LIN {X 0,Y 162.49,Z 738.182,A -85,B 0,C 180,E1 -25157.336,E2 -25157.336} C_VEL
LIN {X 0,Y 169.841,Z 726.293,A -85,B 0,C 180,E1 -25160.422,E2 -25160.422} C_VEL
LIN {X 0,Y 176.479,Z 714.157,A -85,B 0,C 180,E1 -25162.799,E2 -25162.799} C_VEL
LIN {X 0,Y 182.421,Z 701.363,A -85,B 0,C 180,E1 -25164.776,E2 -25164.776} C_VEL
LIN {X 0,Y 187.765,Z 687.719,A -85,B 0,C 180,E1 -25166.394,E2 -25166.394} C_VEL
LIN {X 0,Y 192.387,Z 673.366,A -85,B 0,C 180,E1 -25167.653,E2 -25167.653} C_VEL
LIN {X 0,Y 195.327,Z 661.656,A -85,B 0,C 180,E1 -25168.438,E2 -25168.438} C_VEL
LIN {X 0,Y 188.681,Z 668.85,A -85,B 0,C 180,E1 -25170.426,E2 -25170.426} C_VEL
LIN {X 0,Y 182.829,Z 674.036,A -85,B 0,C 180,E1 -25172.53,E2 -25172.53} C_VEL
LIN {X 0,Y 181.051,Z 675.427,A -85,B 0,C 180,E1 -25173.234,E2 -25173.234} C_VEL
LIN {X 0,Y 174.563,Z 681.994,A -85,B 0,C 180,E1 -25175.551,E2 -25175.551} C_VEL
LIN {X 0,Y 168.965,Z 686.875,A -85,B 0,C 180,E1 -25178.016,E2 -25178.016} C_VEL
LIN {X 0,Y 165.167,Z 689.589,A -85,B 0,C 180,E1 -25180.098,E2 -25180.098} C_VEL
LIN {X 0,Y 163.165,Z 690.902,A -85,B 0,C 180,E1 -25181.38,E2 -25181.38} C_VEL
LIN {X 0,Y 156.436,Z 696.804,A -85,B 0,C 180,E1 -25185.483,E2 -25185.483} C_VEL
LIN {X 0,Y 152.151,Z 700.127,A -85,B 0,C 180,E1 -25189.352,E2 -25189.352} C_VEL
LIN {X 0,Y 149.893,Z 701.971,A -85,B 0,C 180,E1 -25191.914,E2 -25191.914} C_VEL
LIN {X 0,Y 147.571,Z 704.34,A -85,B 0,C 180,E1 -25194.534,E2 -25194.534} C_VEL
LIN {X 0,Y 145.899,Z 706.177,A -85,B 0,C 180,E1 -25197.239,E2 -25197.239} C_VEL
LIN {X 0,Y 143.539,Z 710.381,A -85,B 0,C 180,E1 -25205.619,E2 -25205.619} C_VEL
LIN {X 0,Y 143.347,Z 711.889,A -85,B 0,C 180,E1 -25208.458,E2 -25208.458} C_VEL
LIN {X 0,Y 144.725,Z 713.835,A -85,B 0,C 180,E1 -25214.052,E2 -25214.052} C_VEL
LIN {X 0,Y 149.356,Z 716.433,A -85,B 0,C 180,E1 -25222.113,E2 -25222.113} C_VEL
LIN {X 0,Y 154.656,Z 717.177,A -85,B 0,C 180,E1 -25227.028,E2 -25227.028} C_VEL
LIN {X 0,Y 161.315,Z 717.454,A -85,B 0,C 180,E1 -25231.52,E2 -25231.52} C_VEL
LIN {X 0,Y 168.975,Z 717.586,A -85,B 0,C 180,E1 -25235.611,E2 -25235.611} C_VEL
LIN {X 0,Y 173.986,Z 717.219,A -85,B 0,C 180,E1 -25237.718,E2 -25237.718} C_VEL
LIN {X 0,Y 173.679,Z 718.782,A -85,B 0,C 180,E1 -25238.224,E2 -25238.224} C_VEL
LIN {X 0,Y 167.056,Z 730.388,A -85,B 0,C 180,E1 -25240.773,E2 -25240.773} C_VEL
LIN {X 0,Y 160.359,Z 740.731,A -85,B 0,C 180,E1 -25243.681,E2 -25243.681} C_VEL
LIN {X 0,Y 153.45,Z 750.501,A -85,B 0,C 180,E1 -25247.278,E2 -25247.278} C_VEL
LIN {X 0,Y 147.243,Z 758.709,A -85,B 0,C 180,E1 -25251.245,E2 -25251.245} C_VEL
LIN {X 0,Y 144.176,Z 761.795,A -85,B 0,C 180,E1 -25252.828,E2 -25252.828} C_VEL
LIN {X 0,Y 137.87,Z 766.464,A -85,B 0,C 180,E1 -25255.293,E2 -25255.293} C_VEL
LIN {X 0,Y 131.777,Z 770.674,A -85,B 0,C 180,E1 -25258.095,E2 -25258.095} C_VEL
LIN {X 0,Y 129.133,Z 772.932,A -85,B 0,C 180,E1 -25260.184,E2 -25260.184} C_VEL
LIN {X 0,Y 124.453,Z 778.128,A -85,B 0,C 180,E1 -25266.71,E2 -25266.71} C_VEL
LIN {X 0,Y 121.396,Z 781.651,A -85,B 0,C 180,E1 -25273.169,E2 -25273.169} C_VEL
LIN {X 0,Y 119.749,Z 783.963,A -85,B 0,C 180,E1 -25279.854,E2 -25279.854} C_VEL
LIN {X 0,Y 119.228,Z 785.118,A -85,B 0,C 180,E1 -25286.615,E2 -25286.615} C_VEL
LIN {X 0,Y 119.279,Z 785.267,A -85,B 0,C 180,E1 -25289.995,E2 -25289.995} C_VEL
LIN {X 0,Y 119.386,Z 784.666,A -85,B 0,C 180,E1 -25296.756,E2 -25296.756} C_VEL
LIN {X 0,Y 120.432,Z 782.915,A -85,B 0,C 180,E1 -25303.493,E2 -25303.493} C_VEL
LIN {X 0,Y 122.725,Z 779.989,A -85,B 0,C 180,E1 -25310.09,E2 -25310.09} C_VEL
LIN {X 0,Y 126.443,Z 775.815,A -85,B 0,C 180,E1 -25316.396,E2 -25316.396} C_VEL
LIN {X 0,Y 131.402,Z 770.282,A -85,B 0,C 180,E1 -25322.327,E2 -25322.327} C_VEL
LIN {X 0,Y 137.622,Z 763.238,A -85,B 0,C 180,E1 -25327.787,E2 -25327.787} C_VEL
LIN {X 0,Y 144.102,Z 755.689,A -85,B 0,C 180,E1 -25332.107,E2 -25332.107} C_VEL
LIN {X 0,Y 149.999,Z 747.998,A -85,B 0,C 180,E1 -25335.597,E2 -25335.597} C_VEL
LIN {X 0,Y 157.779,Z 737.318,A -85,B 0,C 180,E1 -25339.214,E2 -25339.214} C_VEL
LIN {X 0,Y 165.444,Z 725.295,A -85,B 0,C 180,E1 -25342.289,E2 -25342.289} C_VEL
LIN {X 0,Y 172.284,Z 713.017,A -85,B 0,C 180,E1 -25344.665,E2 -25344.665} C_VEL
LIN {X 0,Y 178.544,Z 699.747,A -85,B 0,C 180,E1 -25346.657,E2 -25346.657} C_VEL
LIN {X 0,Y 183.943,Z 686.095,A -85,B 0,C 180,E1 -25348.217,E2 -25348.217} C_VEL
LIN {X 0,Y 188.689,Z 671.315,A -85,B 0,C 180,E1 -25349.458,E2 -25349.458} C_VEL
LIN {X 0,Y 192.33,Z 656.608,A -85,B 0,C 180,E1 -25350.334,E2 -25350.334} C_VEL
LIN {X 0,Y 194.901,Z 641.487,A -85,B 0,C 180,E1 -25350.971,E2 -25350.971} C_VEL
LIN {X 0,Y 201.625,Z 569.905,A -85,B 0,C 180,E1 -25352.853,E2 -25352.853} C_VEL
LIN {X 0,Y 204.85,Z 533.822,A -85,B 0,C 180,E1 -25353.826,E2 -25353.826} C_VEL
LIN {X 0,Y 204.843,Z 524.765,A -85,B 0,C 180,E1 -25354.546,E2 -25354.546} C_VEL
LIN {X 0,Y 201.445,Z 518.518,A -85,B 0,C 180,E1 -25357.23,E2 -25357.23} C_VEL
LIN {X 0,Y 196.969,Z 511.105,A -85,B 0,C 180,E1 -25361.404,E2 -25361.404} C_VEL
LIN {X 0,Y 194.313,Z 507.036,A -85,B 0,C 180,E1 -25364.456,E2 -25364.456} C_VEL
LIN {X 0,Y 190.943,Z 502.129,A -85,B 0,C 180,E1 -25369.663,E2 -25369.663} C_VEL
LIN {X 0,Y 189.493,Z 500.135,A -85,B 0,C 180,E1 -25373.077,E2 -25373.077} C_VEL
LIN {X 0,Y 188.395,Z 499.148,A -85,B 0,C 180,E1 -25377.862,E2 -25377.862} C_VEL
LIN {X 0,Y 188.294,Z 499.346,A -85,B 0,C 180,E1 -25381.07,E2 -25381.07} C_VEL
LIN {X 0,Y 188.705,Z 500.765,A -85,B 0,C 180,E1 -25384.564,E2 -25384.564} C_VEL
LIN {X 0,Y 190.134,Z 504.27,A -85,B 0,C 180,E1 -25389.173,E2 -25389.173} C_VEL
LIN {X 0,Y 192.543,Z 509.234,A -85,B 0,C 180,E1 -25393.631,E2 -25393.631} C_VEL
LIN {X 0,Y 195.143,Z 514.935,A -85,B 0,C 180,E1 -25397.172,E2 -25397.172} C_VEL
LIN {X 0,Y 197.823,Z 520.849,A -85,B 0,C 180,E1 -25400.131,E2 -25400.131} C_VEL
LIN {X 0,Y 200.646,Z 527.803,A -85,B 0,C 180,E1 -25402.849,E2 -25402.849} C_VEL
LIN {X 0,Y 203.756,Z 536.057,A -85,B 0,C 180,E1 -25405.5,E2 -25405.5} C_VEL
LIN {X 0,Y 204.496,Z 538.387,A -85,B 0,C 180,E1 -25406.111,E2 -25406.111} C_VEL
LIN {X 0,Y 204.503,Z 541.924,A -85,B 0,C 180,E1 -25406.39,E2 -25406.39} C_VEL
LIN {X 0,Y 195.309,Z 640.75,A -85,B 0,C 180,E1 -25408.979,E2 -25408.979} C_VEL
LIN {X 0,Y 192.93,Z 655.292,A -85,B 0,C 180,E1 -25409.583,E2 -25409.583} C_VEL
LIN {X 0,Y 189.481,Z 669.768,A -85,B 0,C 180,E1 -25410.425,E2 -25410.425} C_VEL
LIN {X 0,Y 185.336,Z 682.994,A -85,B 0,C 180,E1 -25411.446,E2 -25411.446} C_VEL
LIN {X 0,Y 180.038,Z 696.994,A -85,B 0,C 180,E1 -25412.945,E2 -25412.945} C_VEL
LIN {X 0,Y 174.103,Z 710.142,A -85,B 0,C 180,E1 -25414.817,E2 -25414.817} C_VEL
LIN {X 0,Y 167.333,Z 722.659,A -85,B 0,C 180,E1 -25417.067,E2 -25417.067} C_VEL
LIN {X 0,Y 161.275,Z 732.55,A -85,B 0,C 180,E1 -25419.337,E2 -25419.337} C_VEL
LIN {X 0,Y 154.403,Z 742.63,A -85,B 0,C 180,E1 -25422.305,E2 -25422.305} C_VEL
LIN {X 0,Y 146.952,Z 752.624,A -85,B 0,C 180,E1 -25426.215,E2 -25426.215} C_VEL
LIN {X 0,Y 140.359,Z 760.636,A -85,B 0,C 180,E1 -25430.333,E2 -25430.333} C_VEL
LIN {X 0,Y 134.43,Z 767.397,A -85,B 0,C 180,E1 -25434.901,E2 -25434.901} C_VEL
LIN {X 0,Y 128.273,Z 774.274,A -85,B 0,C 180,E1 -25441.239,E2 -25441.239} C_VEL
LIN {X 0,Y 124.469,Z 778.502,A -85,B 0,C 180,E1 -25446.724,E2 -25446.724} C_VEL
LIN {X 0,Y 121.342,Z 782.047,A -85,B 0,C 180,E1 -25453.172,E2 -25453.172} C_VEL
LIN {X 0,Y 119.681,Z 784.387,A -85,B 0,C 180,E1 -25459.859,E2 -25459.859} C_VEL
LIN {X 0,Y 119.151,Z 785.575,A -85,B 0,C 180,E1 -25466.624,E2 -25466.624} C_VEL
LIN {X 0,Y 119.227,Z 785.732,A -85,B 0,C 180,E1 -25470.005,E2 -25470.005} C_VEL
LIN {X 0,Y 119.292,Z 785.153,A -85,B 0,C 180,E1 -25476.772,E2 -25476.772} C_VEL
LIN {X 0,Y 120.374,Z 783.432,A -85,B 0,C 180,E1 -25483.511,E2 -25483.511} C_VEL
LIN {X 0,Y 122.702,Z 780.532,A -85,B 0,C 180,E1 -25490.105,E2 -25490.105} C_VEL
LIN {X 0,Y 126.437,Z 776.387,A -85,B 0,C 180,E1 -25496.408,E2 -25496.408} C_VEL
LIN {X 0,Y 131.398,Z 770.896,A -85,B 0,C 180,E1 -25502.34,E2 -25502.34} C_VEL
LIN {X 0,Y 137.603,Z 763.906,A -85,B 0,C 180,E1 -25507.804,E2 -25507.804} C_VEL
LIN {X 0,Y 144.095,Z 756.412,A -85,B 0,C 180,E1 -25512.121,E2 -25512.121} C_VEL
LIN {X 0,Y 151.1,Z 747.379,A -85,B 0,C 180,E1 -25516.137,E2 -25516.137} C_VEL
LIN {X 0,Y 157.743,Z 738.16,A -85,B 0,C 180,E1 -25519.241,E2 -25519.241} C_VEL
LIN {X 0,Y 165.391,Z 726.268,A -85,B 0,C 180,E1 -25522.325,E2 -25522.325} C_VEL
LIN {X 0,Y 172.271,Z 714.129,A -85,B 0,C 180,E1 -25524.684,E2 -25524.684} C_VEL
LIN {X 0,Y 178.649,Z 700.77,A -85,B 0,C 180,E1 -25526.722,E2 -25526.722} C_VEL
LIN {X 0,Y 184.265,Z 686.688,A -85,B 0,C 180,E1 -25528.345,E2 -25528.345} C_VEL
LIN {X 0,Y 187.983,Z 675.523,A -85,B 0,C 180,E1 -25529.309,E2 -25529.309} C_VEL
LIN {X 0,Y 187.675,Z 675.519,A -85,B 0,C 180,E1 -25529.468,E2 -25529.468} C_VEL
LIN {X 0,Y 180.025,Z 681.759,A -85,B 0,C 180,E1 -25532.065,E2 -25532.065} C_VEL
LIN {X 0,Y 173.593,Z 687.748,A -85,B 0,C 180,E1 -25534.2,E2 -25534.2} C_VEL
LIN {X 0,Y 167.992,Z 692.21,A -85,B 0,C 180,E1 -25536.451,E2 -25536.451} C_VEL
LIN {X 0,Y 163.738,Z 695.116,A -85,B 0,C 180,E1 -25538.602,E2 -25538.602} C_VEL
LIN {X 0,Y 159.607,Z 697.882,A -85,B 0,C 180,E1 -25540.95,E2 -25540.95} C_VEL
LIN {X 0,Y 154.095,Z 702.368,A -85,B 0,C 180,E1 -25544.118,E2 -25544.118} C_VEL
LIN {X 0,Y 148.318,Z 706.43,A -85,B 0,C 180,E1 -25549.074,E2 -25549.074} C_VEL
LIN {X 0,Y 143.513,Z 710.534,A -85,B 0,C 180,E1 -25554.379,E2 -25554.379} C_VEL
LIN {X 0,Y 140.677,Z 713.581,A -85,B 0,C 180,E1 -25560,E2 -25560} C_VEL
LIN {X 0,Y 139.122,Z 717.695,A -85,B 0,C 180,E1 -25568.716,E2 -25568.716} C_VEL
LIN {X 0,Y 140.542,Z 719.536,A -85,B 0,C 180,E1 -25574.479,E2 -25574.479} C_VEL
LIN {X 0,Y 145.295,Z 722.025,A -85,B 0,C 180,E1 -25582.765,E2 -25582.765} C_VEL
LIN {X 0,Y 150.733,Z 722.733,A -85,B 0,C 180,E1 -25587.791,E2 -25587.791} C_VEL
LIN {X 0,Y 161.277,Z 723.193,A -85,B 0,C 180,E1 -25594.507,E2 -25594.507} C_VEL
LIN {X 0,Y 166.326,Z 723.054,A -85,B 0,C 180,E1 -25596.909,E2 -25596.909} C_VEL
LIN {X 0,Y 166.11,Z 724.465,A -85,B 0,C 180,E1 -25597.481,E2 -25597.481} C_VEL
LIN {X 0,Y 158.98,Z 735.806,A -85,B 0,C 180,E1 -25600.304,E2 -25600.304} C_VEL
LIN {X 0,Y 152.197,Z 745.306,A -85,B 0,C 180,E1 -25603.335,E2 -25603.335} C_VEL
LIN {X 0,Y 145.117,Z 754.626,A -85,B 0,C 180,E1 -25607.306,E2 -25607.306} C_VEL
LIN {X 0,Y 138.553,Z 762.37,A -85,B 0,C 180,E1 -25611.578,E2 -25611.578} C_VEL
LIN {X 0,Y 132.923,Z 768.782,A -85,B 0,C 180,E1 -25616.273,E2 -25616.273} C_VEL
LIN {X 0,Y 129.133,Z 772.932,A -85,B 0,C 180,E1 -25620.184,E2 -25620.184} C_VEL
LIN {X 0,Y 126.612,Z 775.054,A -85,B 0,C 180,E1 -25622.385,E2 -25622.385} C_VEL
LIN {X 0,Y 121.161,Z 778.137,A -85,B 0,C 180,E1 -25625.944,E2 -25625.944} C_VEL
LIN {X 0,Y 116.992,Z 780.194,A -85,B 0,C 180,E1 -25629.05,E2 -25629.05} C_VEL
LIN {X 0,Y 114.808,Z 781.484,A -85,B 0,C 180,E1 -25631.694,E2 -25631.694} C_VEL
LIN {X 0,Y 114.384,Z 781.855,A -85,B 0,C 180,E1 -25632.64,E2 -25632.64} C_VEL
LIN {X 0,Y 112.741,Z 783.977,A -85,B 0,C 180,E1 -25639.216,E2 -25639.216} C_VEL
LIN {X 0,Y 112.135,Z 785.132,A -85,B 0,C 180,E1 -25646.401,E2 -25646.401} C_VEL
LIN {X 0,Y 112.198,Z 785.281,A -85,B 0,C 180,E1 -25649.994,E2 -25649.994} C_VEL
LIN {X 0,Y 112.307,Z 784.679,A -85,B 0,C 180,E1 -25657.184,E2 -25657.184} C_VEL
LIN {X 0,Y 113.5,Z 782.929,A -85,B 0,C 180,E1 -25664.335,E2 -25664.335} C_VEL
LIN {X 0,Y 116.051,Z 780.003,A -85,B 0,C 180,E1 -25671.301,E2 -25671.301} C_VEL
LIN {X 0,Y 120.062,Z 775.829,A -85,B 0,C 180,E1 -25677.917,E2 -25677.917} C_VEL
LIN {X 0,Y 125.406,Z 770.296,A -85,B 0,C 180,E1 -25684.078,E2 -25684.078} C_VEL
LIN {X 0,Y 132.036,Z 763.253,A -85,B 0,C 180,E1 -25689.691,E2 -25689.691} C_VEL
LIN {X 0,Y 138.874,Z 755.704,A -85,B 0,C 180,E1 -25694.088,E2 -25694.088} C_VEL
LIN {X 0,Y 143.97,Z 749.356,A -85,B 0,C 180,E1 -25697.067,E2 -25697.067} C_VEL
LIN {X 0,Y 152.012,Z 738.949,A -85,B 0,C 180,E1 -25700.744,E2 -25700.744} C_VEL
LIN {X 0,Y 159.294,Z 728.252,A -85,B 0,C 180,E1 -25703.621,E2 -25703.621} C_VEL
LIN {X 0,Y 166.324,Z 716.568,A -85,B 0,C 180,E1 -25706.014,E2 -25706.014} C_VEL
LIN {X 0,Y 172.742,Z 704.08,A -85,B 0,C 180,E1 -25708.013,E2 -25708.013} C_VEL
LIN {X 0,Y 178.241,Z 691.413,A -85,B 0,C 180,E1 -25709.593,E2 -25709.593} C_VEL
LIN {X 0,Y 183.097,Z 678.132,A -85,B 0,C 180,E1 -25710.829,E2 -25710.829} C_VEL
LIN {X 0,Y 187.313,Z 663.497,A -85,B 0,C 180,E1 -25711.842,E2 -25711.842} C_VEL
LIN {X 0,Y 190.521,Z 648.344,A -85,B 0,C 180,E1 -25712.568,E2 -25712.568} C_VEL
LIN {X 0,Y 192.614,Z 632.59,A -85,B 0,C 180,E1 -25713.075,E2 -25713.075} C_VEL
LIN {X 0,Y 200.135,Z 552.217,A -85,B 0,C 180,E1 -25715.147,E2 -25715.147} C_VEL
LIN {X 0,Y 201.753,Z 534.762,A -85,B 0,C 180,E1 -25715.606,E2 -25715.606} C_VEL
LIN {X 0,Y 201.757,Z 529.052,A -85,B 0,C 180,E1 -25716.092,E2 -25716.092} C_VEL
LIN {X 0,Y 198.348,Z 522.844,A -85,B 0,C 180,E1 -25719.044,E2 -25719.044} C_VEL
LIN {X 0,Y 194.916,Z 516.851,A -85,B 0,C 180,E1 -25722.593,E2 -25722.593} C_VEL
LIN {X 0,Y 192.637,Z 513.263,A -85,B 0,C 180,E1 -25725.439,E2 -25725.439} C_VEL
LIN {X 0,Y 189.566,Z 508.606,A -85,B 0,C 180,E1 -25730.666,E2 -25730.666} C_VEL
LIN {X 0,Y 188.45,Z 507.051,A -85,B 0,C 180,E1 -25733.576,E2 -25733.576} C_VEL
LIN {X 0,Y 187.532,Z 506.19,A -85,B 0,C 180,E1 -25737.852,E2 -25737.852} C_VEL
LIN {X 0,Y 187.425,Z 506.417,A -85,B 0,C 180,E1 -25741.075,E2 -25741.075} C_VEL
LIN {X 0,Y 187.824,Z 507.961,A -85,B 0,C 180,E1 -25744.586,E2 -25744.586} C_VEL
LIN {X 0,Y 189.081,Z 511.235,A -85,B 0,C 180,E1 -25748.82,E2 -25748.82} C_VEL
LIN {X 0,Y 191.124,Z 515.753,A -85,B 0,C 180,E1 -25752.881,E2 -25752.881} C_VEL
LIN {X 0,Y 193.413,Z 521.078,A -85,B 0,C 180,E1 -25756.255,E2 -25756.255} C_VEL
LIN {X 0,Y 195.988,Z 527.127,A -85,B 0,C 180,E1 -25759.312,E2 -25759.312} C_VEL
LIN {X 0,Y 198.545,Z 533.898,A -85,B 0,C 180,E1 -25761.956,E2 -25761.956} C_VEL
LIN {X 0,Y 201.363,Z 541.93,A -85,B 0,C 180,E1 -25764.538,E2 -25764.538} C_VEL
LIN {X 0,Y 196.477,Z 594.889,A -85,B 0,C 180,E1 -25765.947,E2 -25765.947} C_VEL
LIN {X 0,Y 191.811,Z 642.075,A -85,B 0,C 180,E1 -25767.177,E2 -25767.177} C_VEL
LIN {X 0,Y 188.97,Z 657.869,A -85,B 0,C 180,E1 -25767.825,E2 -25767.825} C_VEL
LIN {X 0,Y 184.917,Z 673.444,A -85,B 0,C 180,E1 -25768.783,E2 -25768.783} C_VEL
LIN {X 0,Y 180.361,Z 686.845,A -85,B 0,C 180,E1 -25769.897,E2 -25769.897} C_VEL
LIN {X 0,Y 174.787,Z 700.384,A -85,B 0,C 180,E1 -25771.422,E2 -25771.422} C_VEL
LIN {X 0,Y 168.343,Z 713.578,A -85,B 0,C 180,E1 -25773.396,E2 -25773.396} C_VEL
LIN {X 0,Y 161.206,Z 725.803,A -85,B 0,C 180,E1 -25775.717,E2 -25775.717} C_VEL
LIN {X 0,Y 153.24,Z 737.788,A -85,B 0,C 180,E1 -25778.778,E2 -25778.778} C_VEL
LIN {X 0,Y 145.184,Z 748.444,A -85,B 0,C 180,E1 -25782.428,E2 -25782.428} C_VEL
LIN {X 0,Y 137.965,Z 757.305,A -85,B 0,C 180,E1 -25786.559,E2 -25786.559} C_VEL
LIN {X 0,Y 132.075,Z 763.663,A -85,B 0,C 180,E1 -25790.323,E2 -25790.323} C_VEL
LIN {X 0,Y 125.475,Z 770.703,A -85,B 0,C 180,E1 -25795.943,E2 -25795.943} C_VEL
LIN {X 0,Y 120.137,Z 776.238,A -85,B 0,C 180,E1 -25802.102,E2 -25802.102} C_VEL
LIN {X 0,Y 116.053,Z 780.416,A -85,B 0,C 180,E1 -25808.7,E2 -25808.7} C_VEL
LIN {X 0,Y 113.442,Z 783.35,A -85,B 0,C 180,E1 -25815.658,E2 -25815.658} C_VEL
LIN {X 0,Y 112.241,Z 785.11,A -85,B 0,C 180,E1 -25822.812,E2 -25822.812} C_VEL
LIN {X 0,Y 112.134,Z 785.718,A -85,B 0,C 180,E1 -25830.006,E2 -25830.006} C_VEL
LIN {X 0,Y 112.232,Z 785.139,A -85,B 0,C 180,E1 -25837.2,E2 -25837.2} C_VEL
LIN {X 0,Y 113.427,Z 783.417,A -85,B 0,C 180,E1 -25844.355,E2 -25844.355} C_VEL
LIN {X 0,Y 116.028,Z 780.517,A -85,B 0,C 180,E1 -25851.316,E2 -25851.316} C_VEL
LIN {X 0,Y 120.058,Z 776.371,A -85,B 0,C 180,E1 -25857.93,E2 -25857.93} C_VEL
LIN {X 0,Y 125.398,Z 770.879,A -85,B 0,C 180,E1 -25864.093,E2 -25864.093} C_VEL
LIN {X 0,Y 132.018,Z 763.889,A -85,B 0,C 180,E1 -25869.71,E2 -25869.71} C_VEL
LIN {X 0,Y 138.865,Z 756.393,A -85,B 0,C 180,E1 -25874.104,E2 -25874.104} C_VEL
LIN {X 0,Y 146.233,Z 747.358,A -85,B 0,C 180,E1 -25878.159,E2 -25878.159} C_VEL
LIN {X 0,Y 153.181,Z 738.138,A -85,B 0,C 180,E1 -25881.263,E2 -25881.263} C_VEL
LIN {X 0,Y 161.122,Z 726.243,A -85,B 0,C 180,E1 -25884.337,E2 -25884.337} C_VEL
LIN {X 0,Y 168.264,Z 714.101,A -85,B 0,C 180,E1 -25886.658,E2 -25886.658} C_VEL
LIN {X 0,Y 174.84,Z 700.737,A -85,B 0,C 180,E1 -25888.675,E2 -25888.675} C_VEL
LIN {X 0,Y 179.671,Z 689.175,A -85,B 0,C 180,E1 -25890.002,E2 -25890.002} C_VEL
LIN {X 0,Y 179.716,Z 687.22,A -85,B 0,C 180,E1 -25890.608,E2 -25890.608} C_VEL
LIN {X 0,Y 172.663,Z 693.268,A -85,B 0,C 180,E1 -25892.746,E2 -25892.746} C_VEL
LIN {X 0,Y 166.523,Z 697.794,A -85,B 0,C 180,E1 -25895.036,E2 -25895.036} C_VEL
LIN {X 0,Y 157.57,Z 703.409,A -85,B 0,C 180,E1 -25899.506,E2 -25899.506} C_VEL
LIN {X 0,Y 151.958,Z 707.609,A -85,B 0,C 180,E1 -25902.505,E2 -25902.505} C_VEL
LIN {X 0,Y 144.187,Z 712.624,A -85,B 0,C 180,E1 -25908.757,E2 -25908.757} C_VEL
LIN {X 0,Y 139.219,Z 716.521,A -85,B 0,C 180,E1 -25914.205,E2 -25914.205} C_VEL
LIN {X 0,Y 134.66,Z 722.69,A -85,B 0,C 180,E1 -25927.39,E2 -25927.39} C_VEL
LIN {X 0,Y 135.133,Z 724.293,A -85,B 0,C 180,E1 -25932.007,E2 -25932.007} C_VEL
LIN {X 0,Y 141.041,Z 727.446,A -85,B 0,C 180,E1 -25943.493,E2 -25943.493} C_VEL
LIN {X 0,Y 146.658,Z 728.09,A -85,B 0,C 180,E1 -25948.634,E2 -25948.634} C_VEL
LIN {X 0,Y 158.491,Z 728.513,A -85,B 0,C 180,E1 -25955.973,E2 -25955.973} C_VEL
LIN {X 0,Y 158.11,Z 730.436,A -85,B 0,C 180,E1 -25956.855,E2 -25956.855} C_VEL
LIN {X 0,Y 150.865,Z 740.774,A -85,B 0,C 180,E1 -25959.762,E2 -25959.762} C_VEL
LIN {X 0,Y 143.425,Z 750.353,A -85,B 0,C 180,E1 -25963.315,E2 -25963.315} C_VEL
LIN {X 0,Y 135.959,Z 759.25,A -85,B 0,C 180,E1 -25967.773,E2 -25967.773} C_VEL
LIN {X 0,Y 130.344,Z 765.299,A -85,B 0,C 180,E1 -25971.674,E2 -25971.674} C_VEL
LIN {X 0,Y 124.01,Z 771.915,A -85,B 0,C 180,E1 -25977.42,E2 -25977.42} C_VEL
LIN {X 0,Y 118.932,Z 777.085,A -85,B 0,C 180,E1 -25983.687,E2 -25983.687} C_VEL
LIN {X 0,Y 116.065,Z 780.06,A -85,B 0,C 180,E1 -25988.691,E2 -25988.691} C_VEL
LIN {X 0,Y 114.384,Z 781.855,A -85,B 0,C 180,E1 -25992.64,E2 -25992.64} C_VEL
LIN {X 0,Y 112.854,Z 782.953,A -85,B 0,C 180,E1 -25995.472,E2 -25995.472} C_VEL
LIN {X 0,Y 109.028,Z 784.26,A -85,B 0,C 180,E1 -26000.152,E2 -26000.152} C_VEL
LIN {X 0,Y 106.203,Z 784.924,A -85,B 0,C 180,E1 -26004.121,E2 -26004.121} C_VEL
LIN {X 0,Y 105.086,Z 785.198,A -85,B 0,C 180,E1 -26007.294,E2 -26007.294} C_VEL
LIN {X 0,Y 105.021,Z 785.232,A -85,B 0,C 180,E1 -26008.377,E2 -26008.377} C_VEL
LIN {X 0,Y 105.042,Z 785.14,A -85,B 0,C 180,E1 -26013.83,E2 -26013.83} C_VEL
LIN {X 0,Y 105.753,Z 783.962,A -85,B 0,C 180,E1 -26021.494,E2 -26021.494} C_VEL
LIN {X 0,Y 107.76,Z 781.63,A -85,B 0,C 180,E1 -26029.026,E2 -26029.026} C_VEL
LIN {X 0,Y 111.403,Z 778.092,A -85,B 0,C 180,E1 -26036.2,E2 -26036.2} C_VEL
LIN {X 0,Y 116.489,Z 773.255,A -85,B 0,C 180,E1 -26042.88,E2 -26042.88} C_VEL
LIN {X 0,Y 122.945,Z 766.989,A -85,B 0,C 180,E1 -26048.955,E2 -26048.955} C_VEL
LIN {X 0,Y 129.673,Z 760.223,A -85,B 0,C 180,E1 -26053.704,E2 -26053.704} C_VEL
LIN {X 0,Y 136.401,Z 752.662,A -85,B 0,C 180,E1 -26057.786,E2 -26057.786} C_VEL
LIN {X 0,Y 143.93,Z 743.678,A -85,B 0,C 180,E1 -26061.369,E2 -26061.369} C_VEL
LIN {X 0,Y 151.355,Z 733.848,A -85,B 0,C 180,E1 -26064.342,E2 -26064.342} C_VEL
LIN {X 0,Y 159.109,Z 722.16,A -85,B 0,C 180,E1 -26067.053,E2 -26067.053} C_VEL
LIN {X 0,Y 166.369,Z 709.497,A -85,B 0,C 180,E1 -26069.264,E2 -26069.264} C_VEL
LIN {X 0,Y 172.648,Z 696.361,A -85,B 0,C 180,E1 -26071.06,E2 -26071.06} C_VEL
LIN {X 0,Y 178.293,Z 682.252,A -85,B 0,C 180,E1 -26072.478,E2 -26072.478} C_VEL
LIN {X 0,Y 182.984,Z 667.58,A -85,B 0,C 180,E1 -26073.548,E2 -26073.548} C_VEL
LIN {X 0,Y 186.613,Z 652.278,A -85,B 0,C 180,E1 -26074.348,E2 -26074.348} C_VEL
LIN {X 0,Y 188.971,Z 637.372,A -85,B 0,C 180,E1 -26074.863,E2 -26074.863} C_VEL
LIN {X 0,Y 196.217,Z 563.1,A -85,B 0,C 180,E1 -26076.747,E2 -26076.747} C_VEL
LIN {X 0,Y 198.844,Z 535.581,A -85,B 0,C 180,E1 -26077.461,E2 -26077.461} C_VEL
LIN {X 0,Y 198.833,Z 533.454,A -85,B 0,C 180,E1 -26077.667,E2 -26077.667} C_VEL
LIN {X 0,Y 195.342,Z 526.911,A -85,B 0,C 180,E1 -26081.041,E2 -26081.041} C_VEL
LIN {X 0,Y 192.021,Z 521.025,A -85,B 0,C 180,E1 -26085.02,E2 -26085.02} C_VEL
LIN {X 0,Y 188.697,Z 515.787,A -85,B 0,C 180,E1 -26090.622,E2 -26090.622} C_VEL
LIN {X 0,Y 187.59,Z 514.1,A -85,B 0,C 180,E1 -26093.547,E2 -26093.547} C_VEL
LIN {X 0,Y 186.669,Z 513.23,A -85,B 0,C 180,E1 -26097.843,E2 -26097.843} C_VEL
LIN {X 0,Y 186.558,Z 513.477,A -85,B 0,C 180,E1 -26101.08,E2 -26101.08} C_VEL
LIN {X 0,Y 186.943,Z 515.156,A -85,B 0,C 180,E1 -26104.607,E2 -26104.607} C_VEL
LIN {X 0,Y 188.035,Z 518.201,A -85,B 0,C 180,E1 -26108.463,E2 -26108.463} C_VEL
LIN {X 0,Y 189.77,Z 522.328,A -85,B 0,C 180,E1 -26112.174,E2 -26112.174} C_VEL
LIN {X 0,Y 191.84,Z 527.483,A -85,B 0,C 180,E1 -26115.471,E2 -26115.471} C_VEL
LIN {X 0,Y 194.228,Z 533.508,A -85,B 0,C 180,E1 -26118.521,E2 -26118.521} C_VEL
LIN {X 0,Y 196.953,Z 541.258,A -85,B 0,C 180,E1 -26121.509,E2 -26121.509} C_VEL
LIN {X 0,Y 198.176,Z 545.093,A -85,B 0,C 180,E1 -26122.738,E2 -26122.738} C_VEL
LIN {X 0,Y 197.662,Z 551.323,A -85,B 0,C 180,E1 -26122.955,E2 -26122.955} C_VEL
LIN {X 0,Y 188.839,Z 640.596,A -85,B 0,C 180,E1 -26125.208,E2 -26125.208} C_VEL
LIN {X 0,Y 186.335,Z 655.195,A -85,B 0,C 180,E1 -26125.786,E2 -26125.786} C_VEL
LIN {X 0,Y 182.7,Z 669.696,A -85,B 0,C 180,E1 -26126.582,E2 -26126.582} C_VEL
LIN {X 0,Y 178.334,Z 682.936,A -85,B 0,C 180,E1 -26127.546,E2 -26127.546} C_VEL
LIN {X 0,Y 172.722,Z 696.939,A -85,B 0,C 180,E1 -26128.984,E2 -26128.984} C_VEL
LIN {X 0,Y 166.576,Z 709.688,A -85,B 0,C 180,E1 -26130.708,E2 -26130.708} C_VEL
LIN {X 0,Y 159.808,Z 721.566,A -85,B 0,C 180,E1 -26132.755,E2 -26132.755} C_VEL
LIN {X 0,Y 152.631,Z 732.515,A -85,B 0,C 180,E1 -26135.192,E2 -26135.192} C_VEL
LIN {X 0,Y 145.18,Z 742.597,A -85,B 0,C 180,E1 -26138.135,E2 -26138.135} C_VEL
LIN {X 0,Y 137.126,Z 752.364,A -85,B 0,C 180,E1 -26141.941,E2 -26141.941} C_VEL
LIN {X 0,Y 130.752,Z 759.501,A -85,B 0,C 180,E1 -26145.68,E2 -26145.68} C_VEL
LIN {X 0,Y 124.784,Z 765.574,A -85,B 0,C 180,E1 -26149.639,E2 -26149.639} C_VEL
LIN {X 0,Y 118.025,Z 772.221,A -85,B 0,C 180,E1 -26155.556,E2 -26155.556} C_VEL
LIN {X 0,Y 112.603,Z 777.419,A -85,B 0,C 180,E1 -26162.095,E2 -26162.095} C_VEL
LIN {X 0,Y 109.413,Z 780.402,A -85,B 0,C 180,E1 -26167.338,E2 -26167.338} C_VEL
LIN {X 0,Y 106.529,Z 783.336,A -85,B 0,C 180,E1 -26174.705,E2 -26174.705} C_VEL
LIN {X 0,Y 105.178,Z 785.096,A -85,B 0,C 180,E1 -26182.326,E2 -26182.326} C_VEL
LIN {X 0,Y 105.034,Z 785.704,A -85,B 0,C 180,E1 -26190.006,E2 -26190.006} C_VEL
LIN {X 0,Y 105.172,Z 785.125,A -85,B 0,C 180,E1 -26197.686,E2 -26197.686} C_VEL
LIN {X 0,Y 106.516,Z 783.403,A -85,B 0,C 180,E1 -26205.309,E2 -26205.309} C_VEL
LIN {X 0,Y 109.386,Z 780.502,A -85,B 0,C 180,E1 -26212.681,E2 -26212.681} C_VEL
LIN {X 0,Y 113.775,Z 776.355,A -85,B 0,C 180,E1 -26219.621,E2 -26219.621} C_VEL
LIN {X 0,Y 119.528,Z 770.863,A -85,B 0,C 180,E1 -26226.02,E2 -26226.02} C_VEL
LIN {X 0,Y 126.596,Z 763.871,A -85,B 0,C 180,E1 -26231.779,E2 -26231.779} C_VEL
LIN {X 0,Y 133.803,Z 756.374,A -85,B 0,C 180,E1 -26236.244,E2 -26236.244} C_VEL
LIN {X 0,Y 141.553,Z 747.338,A -85,B 0,C 180,E1 -26240.321,E2 -26240.321} C_VEL
LIN {X 0,Y 148.809,Z 738.116,A -85,B 0,C 180,E1 -26243.412,E2 -26243.412} C_VEL
LIN {X 0,Y 157.079,Z 726.218,A -85,B 0,C 180,E1 -26246.447,E2 -26246.447} C_VEL
LIN {X 0,Y 164.466,Z 714.073,A -85,B 0,C 180,E1 -26248.726,E2 -26248.726} C_VEL
LIN {X 0,Y 171.25,Z 700.703,A -85,B 0,C 180,E1 -26250.708,E2 -26250.708} C_VEL
LIN {X 0,Y 171.706,Z 699.677,A -85,B 0,C 180,E1 -26250.834,E2 -26250.834} C_VEL
LIN {X 0,Y 171.715,Z 698.643,A -85,B 0,C 180,E1 -26251.23,E2 -26251.23} C_VEL
LIN {X 0,Y 164.62,Z 703.489,A -85,B 0,C 180,E1 -26253.713,E2 -26253.713} C_VEL
LIN {X 0,Y 156.425,Z 708.195,A -85,B 0,C 180,E1 -26257.549,E2 -26257.549} C_VEL
LIN {X 0,Y 149.747,Z 712.686,A -85,B 0,C 180,E1 -26260.82,E2 -26260.82} C_VEL
LIN {X 0,Y 142.75,Z 716.801,A -85,B 0,C 180,E1 -26265.749,E2 -26265.749} C_VEL
LIN {X 0,Y 134.058,Z 722.794,A -85,B 0,C 180,E1 -26274.966,E2 -26274.966} C_VEL
LIN {X 0,Y 130,Z 728.744,A -85,B 0,C 180,E1 -26289.333,E2 -26289.333} C_VEL
LIN {X 0,Y 136.622,Z 732.663,A -85,B 0,C 180,E1 -26304.301,E2 -26304.301} C_VEL
LIN {X 0,Y 142.427,Z 733.258,A -85,B 0,C 180,E1 -26309.567,E2 -26309.567} C_VEL
LIN {X 0,Y 150.85,Z 733.573,A -85,B 0,C 180,E1 -26315.036,E2 -26315.036} C_VEL
LIN {X 0,Y 150.988,Z 734.673,A -85,B 0,C 180,E1 -26315.83,E2 -26315.83} C_VEL
LIN {X 0,Y 142.787,Z 745.347,A -85,B 0,C 180,E1 -26319.169,E2 -26319.169} C_VEL
LIN {X 0,Y 134.921,Z 754.664,A -85,B 0,C 180,E1 -26323.17,E2 -26323.17} C_VEL
LIN {X 0,Y 127.672,Z 762.406,A -85,B 0,C 180,E1 -26327.592,E2 -26327.592} C_VEL
LIN {X 0,Y 121.28,Z 768.816,A -85,B 0,C 180,E1 -26332.516,E2 -26332.516} C_VEL
LIN {X 0,Y 115.004,Z 774.76,A -85,B 0,C 180,E1 -26338.82,E2 -26338.82} C_VEL
LIN {X 0,Y 111.417,Z 778.159,A -85,B 0,C 180,E1 -26343.791,E2 -26343.791} C_VEL
LIN {X 0,Y 107.776,Z 781.681,A -85,B 0,C 180,E1 -26350.965,E2 -26350.965} C_VEL
LIN {X 0,Y 105.759,Z 783.991,A -85,B 0,C 180,E1 -26358.495,E2 -26358.495} C_VEL
LIN {X 0,Y 105.043,Z 785.146,A -85,B 0,C 180,E1 -26366.158,E2 -26366.158} C_VEL
LIN {X 0,Y 105.021,Z 785.232,A -85,B 0,C 180,E1 -26368.377,E2 -26368.377} C_VEL
LIN {X 0,Y 104.749,Z 785.278,A -85,B 0,C 180,E1 -26370.514,E2 -26370.514} C_VEL
LIN {X 0,Y 103.979,Z 785.207,A -85,B 0,C 180,E1 -26372.631,E2 -26372.631} C_VEL
LIN {X 0,Y 101.73,Z 784.826,A -85,B 0,C 180,E1 -26376.874,E2 -26376.874} C_VEL
LIN {X 0,Y 99.733,Z 784.146,A -85,B 0,C 180,E1 -26381.301,E2 -26381.301} C_VEL
LIN {X 0,Y 99.341,Z 783.409,A -85,B 0,C 180,E1 -26384.722,E2 -26384.722} C_VEL
LIN {X 0,Y 99.553,Z 783.087,A -85,B 0,C 180,E1 -26385.857,E2 -26385.857} C_VEL
LIN {X 0,Y 102.838,Z 780.03,A -85,B 0,C 180,E1 -26394.201,E2 -26394.201} C_VEL
LIN {X 0,Y 107.61,Z 775.857,A -85,B 0,C 180,E1 -26401.492,E2 -26401.492} C_VEL
LIN {X 0,Y 113.847,Z 770.324,A -85,B 0,C 180,E1 -26408.113,E2 -26408.113} C_VEL
LIN {X 0,Y 121.384,Z 763.282,A -85,B 0,C 180,E1 -26414.002,E2 -26414.002} C_VEL
LIN {X 0,Y 128.946,Z 755.735,A -85,B 0,C 180,E1 -26418.532,E2 -26418.532} C_VEL
LIN {X 0,Y 134.646,Z 749.387,A -85,B 0,C 180,E1 -26421.522,E2 -26421.522} C_VEL
LIN {X 0,Y 143.431,Z 738.982,A -85,B 0,C 180,E1 -26425.15,E2 -26425.15} C_VEL
LIN {X 0,Y 151.278,Z 728.288,A -85,B 0,C 180,E1 -26427.97,E2 -26427.97} C_VEL
LIN {X 0,Y 158.814,Z 716.608,A -85,B 0,C 180,E1 -26430.271,E2 -26430.271} C_VEL
LIN {X 0,Y 165.538,Z 704.345,A -85,B 0,C 180,E1 -26432.16,E2 -26432.16} C_VEL
LIN {X 0,Y 171.49,Z 691.467,A -85,B 0,C 180,E1 -26433.69,E2 -26433.69} C_VEL
LIN {X 0,Y 176.613,Z 678.197,A -85,B 0,C 180,E1 -26434.853,E2 -26434.853} C_VEL
LIN {X 0,Y 181.036,Z 663.582,A -85,B 0,C 180,E1 -26435.814,E2 -26435.814} C_VEL
LIN {X 0,Y 184.399,Z 648.468,A -85,B 0,C 180,E1 -26436.494,E2 -26436.494} C_VEL
LIN {X 0,Y 186.629,Z 632.786,A -85,B 0,C 180,E1 -26436.954,E2 -26436.954} C_VEL
LIN {X 0,Y 194.731,Z 551.1,A -85,B 0,C 180,E1 -26438.974,E2 -26438.974} C_VEL
LIN {X 0,Y 196.026,Z 537.98,A -85,B 0,C 180,E1 -26439.304,E2 -26439.304} C_VEL
LIN {X 0,Y 192.198,Z 530.533,A -85,B 0,C 180,E1 -26443.538,E2 -26443.538} C_VEL
LIN {X 0,Y 190.06,Z 526.801,A -85,B 0,C 180,E1 -26446.485,E2 -26446.485} C_VEL
LIN {X 0,Y 187.486,Z 522.422,A -85,B 0,C 180,E1 -26451.377,E2 -26451.377} C_VEL
LIN {X 0,Y 186.558,Z 521.038,A -85,B 0,C 180,E1 -26454.054,E2 -26454.054} C_VEL
LIN {X 0,Y 185.803,Z 520.287,A -85,B 0,C 180,E1 -26457.832,E2 -26457.832} C_VEL
LIN {X 0,Y 185.69,Z 520.552,A -85,B 0,C 180,E1 -26461.085,E2 -26461.085} C_VEL
LIN {X 0,Y 186.065,Z 522.332,A -85,B 0,C 180,E1 -26464.629,E2 -26464.629} C_VEL
LIN {X 0,Y 187.045,Z 525.285,A -85,B 0,C 180,E1 -26468.236,E2 -26468.236} C_VEL
LIN {X 0,Y 188.479,Z 528.993,A -85,B 0,C 180,E1 -26471.524,E2 -26471.524} C_VEL
LIN {X 0,Y 190.283,Z 533.83,A -85,B 0,C 180,E1 -26474.642,E2 -26474.642} C_VEL
LIN {X 0,Y 192.526,Z 539.929,A -85,B 0,C 180,E1 -26477.738,E2 -26477.738} C_VEL
LIN {X 0,Y 195.236,Z 548.425,A -85,B 0,C 180,E1 -26480.933,E2 -26480.933} C_VEL
LIN {X 0,Y 187.917,Z 622.385,A -85,B 0,C 180,E1 -26482.771,E2 -26482.771} C_VEL
LIN {X 0,Y 185.572,Z 643.223,A -85,B 0,C 180,E1 -26483.317,E2 -26483.317} C_VEL
LIN {X 0,Y 182.592,Z 658.567,A -85,B 0,C 180,E1 -26483.926,E2 -26483.926} C_VEL
LIN {X 0,Y 178.521,Z 673.378,A -85,B 0,C 180,E1 -26484.79,E2 -26484.79} C_VEL
LIN {X 0,Y 173.714,Z 686.788,A -85,B 0,C 180,E1 -26485.829,E2 -26485.829} C_VEL
LIN {X 0,Y 167.949,Z 700.022,A -85,B 0,C 180,E1 -26487.233,E2 -26487.233} C_VEL
LIN {X 0,Y 161.905,Z 711.801,A -85,B 0,C 180,E1 -26488.897,E2 -26488.897} C_VEL
LIN {X 0,Y 154.697,Z 723.657,A -85,B 0,C 180,E1 -26490.971,E2 -26490.971} C_VEL
LIN {X 0,Y 147.322,Z 734.258,A -85,B 0,C 180,E1 -26493.41,E2 -26493.41} C_VEL
LIN {X 0,Y 139.632,Z 744.068,A -85,B 0,C 180,E1 -26496.368,E2 -26496.368} C_VEL
LIN {X 0,Y 131.95,Z 752.888,A -85,B 0,C 180,E1 -26499.89,E2 -26499.89} C_VEL
LIN {X 0,Y 124.655,Z 760.592,A -85,B 0,C 180,E1 -26504.049,E2 -26504.049} C_VEL
LIN {X 0,Y 117.493,Z 767.354,A -85,B 0,C 180,E1 -26508.862,E2 -26508.862} C_VEL
LIN {X 0,Y 110.616,Z 773.621,A -85,B 0,C 180,E1 -26515.131,E2 -26515.131} C_VEL
LIN {X 0,Y 105.061,Z 778.461,A -85,B 0,C 180,E1 -26522.086,E2 -26522.086} C_VEL
LIN {X 0,Y 100.996,Z 782.006,A -85,B 0,C 180,E1 -26529.646,E2 -26529.646} C_VEL
LIN {X 0,Y 98.698,Z 784.346,A -85,B 0,C 180,E1 -26537.672,E2 -26537.672} C_VEL
LIN {X 0,Y 97.887,Z 785.534,A -85,B 0,C 180,E1 -26545.889,E2 -26545.889} C_VEL
LIN {X 0,Y 97.941,Z 785.69,A -85,B 0,C 180,E1 -26550.006,E2 -26550.006} C_VEL
LIN {X 0,Y 98.114,Z 785.11,A -85,B 0,C 180,E1 -26558.243,E2 -26558.243} C_VEL
LIN {X 0,Y 99.647,Z 783.388,A -85,B 0,C 180,E1 -26566.393,E2 -26566.393} C_VEL
LIN {X 0,Y 102.819,Z 780.487,A -85,B 0,C 180,E1 -26574.219,E2 -26574.219} C_VEL
LIN {X 0,Y 107.603,Z 776.339,A -85,B 0,C 180,E1 -26581.507,E2 -26581.507} C_VEL
LIN {X 0,Y 113.822,Z 770.846,A -85,B 0,C 180,E1 -26588.137,E2 -26588.137} C_VEL
LIN {X 0,Y 121.361,Z 763.854,A -85,B 0,C 180,E1 -26594.027,E2 -26594.027} C_VEL
LIN {X 0,Y 128.945,Z 756.355,A -85,B 0,C 180,E1 -26598.547,E2 -26598.547} C_VEL
LIN {X 0,Y 137.109,Z 747.317,A -85,B 0,C 180,E1 -26602.615,E2 -26602.615} C_VEL
LIN {X 0,Y 144.678,Z 738.094,A -85,B 0,C 180,E1 -26605.677,E2 -26605.677} C_VEL
LIN {X 0,Y 153.261,Z 726.193,A -85,B 0,C 180,E1 -26608.664,E2 -26608.664} C_VEL
LIN {X 0,Y 160.886,Z 714.044,A -85,B 0,C 180,E1 -26610.893,E2 -26610.893} C_VEL
LIN {X 0,Y 163.922,Z 708.301,A -85,B 0,C 180,E1 -26611.861,E2 -26611.861} C_VEL
LIN {X 0,Y 156.795,Z 712.131,A -85,B 0,C 180,E1 -26614.797,E2 -26614.797} C_VEL
LIN {X 0,Y 152.399,Z 714.663,A -85,B 0,C 180,E1 -26616.778,E2 -26616.778} C_VEL
LIN {X 0,Y 145.419,Z 718.846,A -85,B 0,C 180,E1 -26620.226,E2 -26620.226} C_VEL
LIN {X 0,Y 132.309,Z 726.316,A -85,B 0,C 180,E1 -26630.83,E2 -26630.83} C_VEL
LIN {X 0,Y 128.117,Z 729.229,A -85,B 0,C 180,E1 -26636.855,E2 -26636.855} C_VEL
LIN {X 0,Y 125.117,Z 733.972,A -85,B 0,C 180,E1 -26649.701,E2 -26649.701} C_VEL
LIN {X 0,Y 132.052,Z 737.671,A -85,B 0,C 180,E1 -26665.199,E2 -26665.199} C_VEL
LIN {X 0,Y 138.055,Z 738.231,A -85,B 0,C 180,E1 -26670.602,E2 -26670.602} C_VEL
LIN {X 0,Y 142.995,Z 738.344,A -85,B 0,C 180,E1 -26673.91,E2 -26673.91} C_VEL
LIN {X 0,Y 143.626,Z 739.002,A -85,B 0,C 180,E1 -26674.793,E2 -26674.793} C_VEL
LIN {X 0,Y 135.947,Z 748.229,A -85,B 0,C 180,E1 -26677.96,E2 -26677.96} C_VEL
LIN {X 0,Y 127.931,Z 757.071,A -85,B 0,C 180,E1 -26682.123,E2 -26682.123} C_VEL
LIN {X 0,Y 119.434,Z 765.334,A -85,B 0,C 180,E1 -26687.406,E2 -26687.406} C_VEL
LIN {X 0,Y 112.219,Z 771.948,A -85,B 0,C 180,E1 -26693.484,E2 -26693.484} C_VEL
LIN {X 0,Y 106.299,Z 777.116,A -85,B 0,C 180,E1 -26700.267,E2 -26700.267} C_VEL
LIN {X 0,Y 102.852,Z 780.091,A -85,B 0,C 180,E1 -26705.79,E2 -26705.79} C_VEL
LIN {X 0,Y 99.713,Z 782.998,A -85,B 0,C 180,E1 -26713.618,E2 -26713.618} C_VEL
LIN {X 0,Y 98.203,Z 784.725,A -85,B 0,C 180,E1 -26721.765,E2 -26721.765} C_VEL
LIN {X 0,Y 98.005,Z 785.309,A -85,B 0,C 180,E1 -26729.994,E2 -26729.994} C_VEL
LIN {X 0,Y 98.2,Z 784.707,A -85,B 0,C 180,E1 -26738.223,E2 -26738.223} C_VEL
LIN {X 0,Y 99.553,Z 783.087,A -85,B 0,C 180,E1 -26745.857,E2 -26745.857} C_VEL
LIN {X 0,Y 99.963,Z 782.155,A -85,B 0,C 180,E1 -26749.194,E2 -26749.194} C_VEL
LIN {X 0,Y 99.505,Z 780.235,A -85,B 0,C 180,E1 -26754.772,E2 -26754.772} C_VEL
LIN {X 0,Y 99.577,Z 778.317,A -85,B 0,C 180,E1 -26759.223,E2 -26759.223} C_VEL
LIN {X 0,Y 100.71,Z 776.654,A -85,B 0,C 180,E1 -26762.41,E2 -26762.41} C_VEL
LIN {X 0,Y 101.389,Z 776.005,A -85,B 0,C 180,E1 -26763.402,E2 -26763.402} C_VEL
LIN {X 0,Y 108.315,Z 770.338,A -85,B 0,C 180,E1 -26770.446,E2 -26770.446} C_VEL
LIN {X 0,Y 116.349,Z 763.296,A -85,B 0,C 180,E1 -26776.448,E2 -26776.448} C_VEL
LIN {X 0,Y 123.172,Z 756.932,A -85,B 0,C 180,E1 -26780.371,E2 -26780.371} C_VEL
LIN {X 0,Y 130.337,Z 749.403,A -85,B 0,C 180,E1 -26783.972,E2 -26783.972} C_VEL
LIN {X 0,Y 139.481,Z 738.999,A -85,B 0,C 180,E1 -26787.553,E2 -26787.553} C_VEL
LIN {X 0,Y 147.616,Z 728.306,A -85,B 0,C 180,E1 -26790.319,E2 -26790.319} C_VEL
LIN {X 0,Y 155.407,Z 716.628,A -85,B 0,C 180,E1 -26792.551,E2 -26792.551} C_VEL
LIN {X 0,Y 162.563,Z 703.914,A -85,B 0,C 180,E1 -26794.445,E2 -26794.445} C_VEL
LIN {X 0,Y 168.46,Z 691.493,A -85,B 0,C 180,E1 -26795.857,E2 -26795.857} C_VEL
LIN {X 0,Y 174.094,Z 677.124,A -85,B 0,C 180,E1 -26797.05,E2 -26797.05} C_VEL
LIN {X 0,Y 178.64,Z 662.141,A -85,B 0,C 180,E1 -26797.959,E2 -26797.959} C_VEL
LIN {X 0,Y 182.075,Z 646.339,A -85,B 0,C 180,E1 -26798.613,E2 -26798.613} C_VEL
LIN {X 0,Y 184.338,Z 629.346,A -85,B 0,C 180,E1 -26799.068,E2 -26799.068} C_VEL
LIN {X 0,Y 193.098,Z 543.484,A -85,B 0,C 180,E1 -26801.125,E2 -26801.125} C_VEL
LIN {X 0,Y 193.186,Z 542.18,A -85,B 0,C 180,E1 -26801.196,E2 -26801.196} C_VEL
LIN {X 0,Y 190.322,Z 536.333,A -85,B 0,C 180,E1 -26804.746,E2 -26804.746} C_VEL
LIN {X 0,Y 188.512,Z 533.095,A -85,B 0,C 180,E1 -26807.485,E2 -26807.485} C_VEL
LIN {X 0,Y 186.303,Z 529.103,A -85,B 0,C 180,E1 -26812.141,E2 -26812.141} C_VEL
LIN {X 0,Y 185.541,Z 527.971,A -85,B 0,C 180,E1 -26814.566,E2 -26814.566} C_VEL
LIN {X 0,Y 184.937,Z 527.344,A -85,B 0,C 180,E1 -26817.822,E2 -26817.822} C_VEL
LIN {X 0,Y 184.821,Z 527.63,A -85,B 0,C 180,E1 -26821.09,E2 -26821.09} C_VEL
LIN {X 0,Y 185.185,Z 529.521,A -85,B 0,C 180,E1 -26824.651,E2 -26824.651} C_VEL
LIN {X 0,Y 186.198,Z 532.785,A -85,B 0,C 180,E1 -26828.411,E2 -26828.411} C_VEL
LIN {X 0,Y 187.247,Z 535.709,A -85,B 0,C 180,E1 -26830.929,E2 -26830.929} C_VEL
LIN {X 0,Y 188.826,Z 540.391,A -85,B 0,C 180,E1 -26833.904,E2 -26833.904} C_VEL
LIN {X 0,Y 190.691,Z 545.882,A -85,B 0,C 180,E1 -26836.713,E2 -26836.713} C_VEL
LIN {X 0,Y 192.479,Z 551.875,A -85,B 0,C 180,E1 -26839.072,E2 -26839.072} C_VEL
LIN {X 0,Y 183.432,Z 639.032,A -85,B 0,C 180,E1 -26841.151,E2 -26841.151} C_VEL
LIN {X 0,Y 180.795,Z 654.214,A -85,B 0,C 180,E1 -26841.685,E2 -26841.685} C_VEL
LIN {X 0,Y 177.18,Z 668.36,A -85,B 0,C 180,E1 -26842.387,E2 -26842.387} C_VEL
LIN {X 0,Y 172.234,Z 682.877,A -85,B 0,C 180,E1 -26843.359,E2 -26843.359} C_VEL
LIN {X 0,Y 166.287,Z 696.89,A -85,B 0,C 180,E1 -26844.687,E2 -26844.687} C_VEL
LIN {X 0,Y 159.349,Z 710.401,A -85,B 0,C 180,E1 -26846.427,E2 -26846.427} C_VEL
LIN {X 0,Y 151.868,Z 722.583,A -85,B 0,C 180,E1 -26848.456,E2 -26848.456} C_VEL
LIN {X 0,Y 143.512,Z 734.241,A -85,B 0,C 180,E1 -26851.028,E2 -26851.028} C_VEL
LIN {X 0,Y 135.517,Z 744.052,A -85,B 0,C 180,E1 -26853.934,E2 -26853.934} C_VEL
LIN {X 0,Y 126.941,Z 753.412,A -85,B 0,C 180,E1 -26857.681,E2 -26857.681} C_VEL
LIN {X 0,Y 119.806,Z 760.578,A -85,B 0,C 180,E1 -26861.597,E2 -26861.597} C_VEL
LIN {X 0,Y 112.201,Z 767.34,A -85,B 0,C 180,E1 -26866.457,E2 -26866.457} C_VEL
LIN {X 0,Y 104.81,Z 773.607,A -85,B 0,C 180,E1 -26872.888,E2 -26872.888} C_VEL
LIN {X 0,Y 98.799,Z 778.448,A -85,B 0,C 180,E1 -26880.144,E2 -26880.144} C_VEL
LIN {X 0,Y 94.324,Z 781.992,A -85,B 0,C 180,E1 -26888.135,E2 -26888.135} C_VEL
LIN {X 0,Y 91.754,Z 784.332,A -85,B 0,C 180,E1 -26896.723,E2 -26896.723} C_VEL
LIN {X 0,Y 90.799,Z 785.52,A -85,B 0,C 180,E1 -26905.568,E2 -26905.568} C_VEL
LIN {X 0,Y 90.841,Z 785.677,A -85,B 0,C 180,E1 -26910.007,E2 -26910.007} C_VEL
LIN {X 0,Y 91.082,Z 785.096,A -85,B 0,C 180,E1 -26918.884,E2 -26918.884} C_VEL
LIN {X 0,Y 92.827,Z 783.373,A -85,B 0,C 180,E1 -26927.635,E2 -26927.635} C_VEL
LIN {X 0,Y 96.343,Z 780.471,A -85,B 0,C 180,E1 -26935.963,E2 -26935.963} C_VEL
LIN {X 0,Y 102.05,Z 775.894,A -85,B 0,C 180,E1 -26944.266,E2 -26944.266} C_VEL
LIN {X 0,Y 108.267,Z 770.83,A -85,B 0,C 180,E1 -26950.483,E2 -26950.483} C_VEL
LIN {X 0,Y 116.335,Z 763.836,A -85,B 0,C 180,E1 -26956.471,E2 -26956.471} C_VEL
LIN {X 0,Y 124.311,Z 756.336,A -85,B 0,C 180,E1 -26961.027,E2 -26961.027} C_VEL
LIN {X 0,Y 132.897,Z 747.297,A -85,B 0,C 180,E1 -26965.061,E2 -26965.061} C_VEL
LIN {X 0,Y 140.778,Z 738.072,A -85,B 0,C 180,E1 -26968.076,E2 -26968.076} C_VEL
LIN {X 0,Y 149.677,Z 726.168,A -85,B 0,C 180,E1 -26970.996,E2 -26970.996} C_VEL
LIN {X 0,Y 154.664,Z 718.654,A -85,B 0,C 180,E1 -26972.393,E2 -26972.393} C_VEL
LIN {X 0,Y 155.029,Z 717.163,A -85,B 0,C 180,E1 -26973.042,E2 -26973.042} C_VEL
LIN {X 0,Y 150.187,Z 719.724,A -85,B 0,C 180,E1 -26975.092,E2 -26975.092} C_VEL
LIN {X 0,Y 144.389,Z 722.949,A -85,B 0,C 180,E1 -26977.649,E2 -26977.649} C_VEL
LIN {X 0,Y 137.085,Z 726.586,A -85,B 0,C 180,E1 -26982.085,E2 -26982.085} C_VEL
LIN {X 0,Y 127.384,Z 731.789,A -85,B 0,C 180,E1 -26990.473,E2 -26990.473} C_VEL
LIN {X 0,Y 121.715,Z 735.657,A -85,B 0,C 180,E1 -27000,E2 -27000} C_VEL
LIN {X 0,Y 120.061,Z 738.029,A -85,B 0,C 180,E1 -27006.723,E2 -27006.723} C_VEL
LIN {X 0,Y 121.699,Z 740.461,A -85,B 0,C 180,E1 -27016.783,E2 -27016.783} C_VEL
LIN {X 0,Y 127.324,Z 742.475,A -85,B 0,C 180,E1 -27026.204,E2 -27026.204} C_VEL
LIN {X 0,Y 133.569,Z 742.987,A -85,B 0,C 180,E1 -27031.747,E2 -27031.747} C_VEL
LIN {X 0,Y 135.531,Z 743.917,A -85,B 0,C 180,E1 -27033.927,E2 -27033.927} C_VEL
LIN {X 0,Y 127.026,Z 753.193,A -85,B 0,C 180,E1 -27037.65,E2 -27037.65} C_VEL
LIN {X 0,Y 118.661,Z 761.441,A -85,B 0,C 180,E1 -27042.232,E2 -27042.232} C_VEL
LIN {X 0,Y 110.25,Z 768.849,A -85,B 0,C 180,E1 -27047.977,E2 -27047.977} C_VEL
LIN {X 0,Y 102.954,Z 774.842,A -85,B 0,C 180,E1 -27054.766,E2 -27054.766} C_VEL
LIN {X 0,Y 98.773,Z 778.19,A -85,B 0,C 180,E1 -27060.121,E2 -27060.121} C_VEL
LIN {X 0,Y 94.362,Z 781.711,A -85,B 0,C 180,E1 -27068.13,E2 -27068.13} C_VEL
LIN {X 0,Y 91.818,Z 784.02,A -85,B 0,C 180,E1 -27076.718,E2 -27076.718} C_VEL
LIN {X 0,Y 90.877,Z 785.174,A -85,B 0,C 180,E1 -27085.558,E2 -27085.558} C_VEL
LIN {X 0,Y 90.912,Z 785.322,A -85,B 0,C 180,E1 -27089.993,E2 -27089.993} C_VEL
LIN {X 0,Y 91.152,Z 784.721,A -85,B 0,C 180,E1 -27098.864,E2 -27098.864} C_VEL
LIN {X 0,Y 92.872,Z 782.97,A -85,B 0,C 180,E1 -27107.612,E2 -27107.612} C_VEL
LIN {X 0,Y 96.358,Z 780.044,A -85,B 0,C 180,E1 -27115.944,E2 -27115.944} C_VEL
LIN {X 0,Y 101.389,Z 776.005,A -85,B 0,C 180,E1 -27123.402,E2 -27123.402} C_VEL
LIN {X 0,Y 103.2,Z 774.105,A -85,B 0,C 180,E1 -27126.371,E2 -27126.371} C_VEL
LIN {X 0,Y 105.136,Z 770.723,A -85,B 0,C 180,E1 -27131.4,E2 -27131.4} C_VEL
LIN {X 0,Y 107.756,Z 766.866,A -85,B 0,C 180,E1 -27136.11,E2 -27136.11} C_VEL
LIN {X 0,Y 110.504,Z 764.19,A -85,B 0,C 180,E1 -27138.465,E2 -27138.465} C_VEL
LIN {X 0,Y 118.721,Z 756.947,A -85,B 0,C 180,E1 -27143.041,E2 -27143.041} C_VEL
LIN {X 0,Y 126.274,Z 749.418,A -85,B 0,C 180,E1 -27146.59,E2 -27146.59} C_VEL
LIN {X 0,Y 135.778,Z 739.015,A -85,B 0,C 180,E1 -27150.101,E2 -27150.101} C_VEL
LIN {X 0,Y 144.226,Z 728.324,A -85,B 0,C 180,E1 -27152.775,E2 -27152.775} C_VEL
LIN {X 0,Y 152.249,Z 716.648,A -85,B 0,C 180,E1 -27154.935,E2 -27154.935} C_VEL
LIN {X 0,Y 159.4,Z 704.358,A -85,B 0,C 180,E1 -27156.697,E2 -27156.697} C_VEL
LIN {X 0,Y 165.687,Z 691.519,A -85,B 0,C 180,E1 -27158.094,E2 -27158.094} C_VEL
LIN {X 0,Y 171.447,Z 677.156,A -85,B 0,C 180,E1 -27159.238,E2 -27159.238} C_VEL
LIN {X 0,Y 176.103,Z 662.184,A -85,B 0,C 180,E1 -27160.097,E2 -27160.097} C_VEL
LIN {X 0,Y 179.61,Z 646.403,A -85,B 0,C 180,E1 -27160.721,E2 -27160.721} C_VEL
LIN {X 0,Y 181.93,Z 629.448,A -85,B 0,C 180,E1 -27161.15,E2 -27161.15} C_VEL
LIN {X 0,Y 190.451,Z 548.14,A -85,B 0,C 180,E1 -27163.029,E2 -27163.029} C_VEL
LIN {X 0,Y 190.564,Z 546.574,A -85,B 0,C 180,E1 -27163.116,E2 -27163.116} C_VEL
LIN {X 0,Y 188.288,Z 541.668,A -85,B 0,C 180,E1 -27166.355,E2 -27166.355} C_VEL
LIN {X 0,Y 185.783,Z 537.012,A -85,B 0,C 180,E1 -27171.16,E2 -27171.16} C_VEL
LIN {X 0,Y 184.832,Z 535.191,A -85,B 0,C 180,E1 -27173.998,E2 -27173.998} C_VEL
LIN {X 0,Y 184.071,Z 534.401,A -85,B 0,C 180,E1 -27177.812,E2 -27177.812} C_VEL
LIN {X 0,Y 183.954,Z 534.69,A -85,B 0,C 180,E1 -27181.095,E2 -27181.095} C_VEL
LIN {X 0,Y 184.346,Z 536.931,A -85,B 0,C 180,E1 -27184.921,E2 -27184.921} C_VEL
LIN {X 0,Y 185.66,Z 541.185,A -85,B 0,C 180,E1 -27189.396,E2 -27189.396} C_VEL
LIN {X 0,Y 187.197,Z 546.252,A -85,B 0,C 180,E1 -27192.77,E2 -27192.77} C_VEL
LIN {X 0,Y 188.919,Z 551.794,A -85,B 0,C 180,E1 -27195.664,E2 -27195.664} C_VEL
LIN {X 0,Y 189.884,Z 555.424,A -85,B 0,C 180,E1 -27197.125,E2 -27197.125} C_VEL
LIN {X 0,Y 180.977,Z 639.102,A -85,B 0,C 180,E1 -27199.064,E2 -27199.064} C_VEL
LIN {X 0,Y 178.285,Z 654.165,A -85,B 0,C 180,E1 -27199.557,E2 -27199.557} C_VEL
LIN {X 0,Y 174.6,Z 668.323,A -85,B 0,C 180,E1 -27200.232,E2 -27200.232} C_VEL
LIN {X 0,Y 169.539,Z 682.847,A -85,B 0,C 180,E1 -27201.152,E2 -27201.152} C_VEL
LIN {X 0,Y 163.442,Z 696.865,A -85,B 0,C 180,E1 -27202.419,E2 -27202.419} C_VEL
LIN {X 0,Y 157.192,Z 708.849,A -85,B 0,C 180,E1 -27203.863,E2 -27203.863} C_VEL
LIN {X 0,Y 149.346,Z 721.51,A -85,B 0,C 180,E1 -27205.854,E2 -27205.854} C_VEL
LIN {X 0,Y 141.392,Z 732.462,A -85,B 0,C 180,E1 -27208.093,E2 -27208.093} C_VEL
LIN {X 0,Y 133.04,Z 742.549,A -85,B 0,C 180,E1 -27210.87,E2 -27210.87} C_VEL
LIN {X 0,Y 123.272,Z 752.835,A -85,B 0,C 180,E1 -27214.759,E2 -27214.759} C_VEL
LIN {X 0,Y 115.187,Z 760.563,A -85,B 0,C 180,E1 -27218.939,E2 -27218.939} C_VEL
LIN {X 0,Y 107.12,Z 767.326,A -85,B 0,C 180,E1 -27223.815,E2 -27223.815} C_VEL
LIN {X 0,Y 99.187,Z 773.593,A -85,B 0,C 180,E1 -27230.388,E2 -27230.388} C_VEL
LIN {X 0,Y 92.671,Z 778.434,A -85,B 0,C 180,E1 -27237.944,E2 -27237.944} C_VEL
LIN {X 0,Y 87.731,Z 781.978,A -85,B 0,C 180,E1 -27246.396,E2 -27246.396} C_VEL
LIN {X 0,Y 84.819,Z 784.319,A -85,B 0,C 180,E1 -27255.614,E2 -27255.614} C_VEL
LIN {X 0,Y 83.714,Z 785.506,A -85,B 0,C 180,E1 -27265.192,E2 -27265.192} C_VEL
LIN {X 0,Y 83.762,Z 785.663,A -85,B 0,C 180,E1 -27270.007,E2 -27270.007} C_VEL
LIN {X 0,Y 84.049,Z 785.082,A -85,B 0,C 180,E1 -27279.635,E2 -27279.635} C_VEL
LIN {X 0,Y 86.042,Z 783.359,A -85,B 0,C 180,E1 -27289.077,E2 -27289.077} C_VEL
LIN {X 0,Y 89.974,Z 780.456,A -85,B 0,C 180,E1 -27297.955,E2 -27297.955} C_VEL
LIN {X 0,Y 95.807,Z 776.183,A -85,B 0,C 180,E1 -27306.204,E2 -27306.204} C_VEL
LIN {X 0,Y 102.928,Z 770.813,A -85,B 0,C 180,E1 -27313.071,E2 -27313.071} C_VEL
LIN {X 0,Y 111.547,Z 763.818,A -85,B 0,C 180,E1 -27319.126,E2 -27319.126} C_VEL
LIN {X 0,Y 119.926,Z 756.317,A -85,B 0,C 180,E1 -27323.694,E2 -27323.694} C_VEL
LIN {X 0,Y 128.935,Z 747.276,A -85,B 0,C 180,E1 -27327.667,E2 -27327.667} C_VEL
LIN {X 0,Y 137.133,Z 738.05,A -85,B 0,C 180,E1 -27330.611,E2 -27330.611} C_VEL
LIN {X 0,Y 145.634,Z 727.118,A -85,B 0,C 180,E1 -27333.232,E2 -27333.232} C_VEL
LIN {X 0,Y 146.421,Z 725.451,A -85,B 0,C 180,E1 -27333.898,E2 -27333.898} C_VEL
LIN {X 0,Y 140.62,Z 728.334,A -85,B 0,C 180,E1 -27336.432,E2 -27336.432} C_VEL
LIN {X 0,Y 132.292,Z 732.102,A -85,B 0,C 180,E1 -27341.412,E2 -27341.412} C_VEL
LIN {X 0,Y 120.646,Z 737.895,A -85,B 0,C 180,E1 -27352.045,E2 -27352.045} C_VEL
LIN {X 0,Y 114.764,Z 742.888,A -85,B 0,C 180,E1 -27367.035,E2 -27367.035} C_VEL
LIN {X 0,Y 116.524,Z 745.172,A -85,B 0,C 180,E1 -27377.551,E2 -27377.551} C_VEL
LIN {X 0,Y 122.468,Z 747.037,A -85,B 0,C 180,E1 -27387.328,E2 -27387.328} C_VEL
LIN {X 0,Y 127.83,Z 747.476,A -85,B 0,C 180,E1 -27392.156,E2 -27392.156} C_VEL
LIN {X 0,Y 127.009,Z 748.926,A -85,B 0,C 180,E1 -27393.159,E2 -27393.159} C_VEL
LIN {X 0,Y 118.799,Z 757.108,A -85,B 0,C 180,E1 -27396.991,E2 -27396.991} C_VEL
LIN {X 0,Y 111.595,Z 763.459,A -85,B 0,C 180,E1 -27400.903,E2 -27400.903} C_VEL
LIN {X 0,Y 103.008,Z 770.465,A -85,B 0,C 180,E1 -27406.971,E2 -27406.971} C_VEL
LIN {X 0,Y 95.701,Z 775.967,A -85,B 0,C 180,E1 -27414.013,E2 -27414.013} C_VEL
LIN {X 0,Y 90.001,Z 780.121,A -85,B 0,C 180,E1 -27422.054,E2 -27422.054} C_VEL
LIN {X 0,Y 86.095,Z 783.027,A -85,B 0,C 180,E1 -27430.935,E2 -27430.935} C_VEL
LIN {X 0,Y 84.136,Z 784.753,A -85,B 0,C 180,E1 -27440.376,E2 -27440.376} C_VEL
LIN {X 0,Y 83.811,Z 785.336,A -85,B 0,C 180,E1 -27449.993,E2 -27449.993} C_VEL
LIN {X 0,Y 84.132,Z 784.734,A -85,B 0,C 180,E1 -27459.61,E2 -27459.61} C_VEL
LIN {X 0,Y 86.082,Z 782.984,A -85,B 0,C 180,E1 -27469.053,E2 -27469.053} C_VEL
LIN {X 0,Y 89.986,Z 780.057,A -85,B 0,C 180,E1 -27477.936,E2 -27477.936} C_VEL
LIN {X 0,Y 96.05,Z 775.608,A -85,B 0,C 180,E1 -27486.403,E2 -27486.403} C_VEL
LIN {X 0,Y 102.961,Z 770.352,A -85,B 0,C 180,E1 -27493.037,E2 -27493.037} C_VEL
LIN {X 0,Y 110.504,Z 764.19,A -85,B 0,C 180,E1 -27498.465,E2 -27498.465} C_VEL
LIN {X 0,Y 113.365,Z 761.387,A -85,B 0,C 180,E1 -27500.687,E2 -27500.687} C_VEL
LIN {X 0,Y 116.919,Z 756.662,A -85,B 0,C 180,E1 -27504.658,E2 -27504.658} C_VEL
LIN {X 0,Y 120.775,Z 751.502,A -85,B 0,C 180,E1 -27508.291,E2 -27508.291} C_VEL
LIN {X 0,Y 123.956,Z 747.997,A -85,B 0,C 180,E1 -27509.94,E2 -27509.94} C_VEL
LIN {X 0,Y 133.804,Z 737.42,A -85,B 0,C 180,E1 -27513.23,E2 -27513.23} C_VEL
LIN {X 0,Y 143.35,Z 725.407,A -85,B 0,C 180,E1 -27515.928,E2 -27515.928} C_VEL
LIN {X 0,Y 151.657,Z 713.142,A -85,B 0,C 180,E1 -27517.933,E2 -27517.933} C_VEL
LIN {X 0,Y 158.525,Z 701.088,A -85,B 0,C 180,E1 -27519.466,E2 -27519.466} C_VEL
LIN {X 0,Y 164.733,Z 688.075,A -85,B 0,C 180,E1 -27520.706,E2 -27520.706} C_VEL
LIN {X 0,Y 170.248,Z 673.878,A -85,B 0,C 180,E1 -27521.692,E2 -27521.692} C_VEL
LIN {X 0,Y 174.619,Z 659.265,A -85,B 0,C 180,E1 -27522.419,E2 -27522.419} C_VEL
LIN {X 0,Y 177.79,Z 644.282,A -85,B 0,C 180,E1 -27522.951,E2 -27522.951} C_VEL
LIN {X 0,Y 180.347,Z 624.187,A -85,B 0,C 180,E1 -27523.401,E2 -27523.401} C_VEL
LIN {X 0,Y 188.077,Z 552.116,A -85,B 0,C 180,E1 -27525.018,E2 -27525.018} C_VEL
LIN {X 0,Y 188.158,Z 551.018,A -85,B 0,C 180,E1 -27525.085,E2 -27525.085} C_VEL
LIN {X 0,Y 186.292,Z 547.015,A -85,B 0,C 180,E1 -27528.163,E2 -27528.163} C_VEL
LIN {X 0,Y 184.24,Z 542.843,A -85,B 0,C 180,E1 -27533.016,E2 -27533.016} C_VEL
LIN {X 0,Y 183.55,Z 541.838,A -85,B 0,C 180,E1 -27535.608,E2 -27535.608} C_VEL
LIN {X 0,Y 183.205,Z 541.458,A -85,B 0,C 180,E1 -27537.802,E2 -27537.802} C_VEL
LIN {X 0,Y 183.083,Z 541.781,A -85,B 0,C 180,E1 -27541.1,E2 -27541.1} C_VEL
LIN {X 0,Y 183.532,Z 544.439,A -85,B 0,C 180,E1 -27545.303,E2 -27545.303} C_VEL
LIN {X 0,Y 184.631,Z 548.49,A -85,B 0,C 180,E1 -27549.172,E2 -27549.172} C_VEL
LIN {X 0,Y 185.821,Z 552.812,A -85,B 0,C 180,E1 -27552.006,E2 -27552.006} C_VEL
LIN {X 0,Y 187.137,Z 557.49,A -85,B 0,C 180,E1 -27554.476,E2 -27554.476} C_VEL
LIN {X 0,Y 187.519,Z 559.032,A -85,B 0,C 180,E1 -27555.14,E2 -27555.14} C_VEL
LIN {X 0,Y 178.645,Z 640.016,A -85,B 0,C 180,E1 -27556.937,E2 -27556.937} C_VEL
LIN {X 0,Y 175.842,Z 654.995,A -85,B 0,C 180,E1 -27557.417,E2 -27557.417} C_VEL
LIN {X 0,Y 171.884,Z 669.55,A -85,B 0,C 180,E1 -27558.09,E2 -27558.09} C_VEL
LIN {X 0,Y 167.11,Z 682.819,A -85,B 0,C 180,E1 -27558.883,E2 -27558.883} C_VEL
LIN {X 0,Y 160.864,Z 696.841,A -85,B 0,C 180,E1 -27560.077,E2 -27560.077} C_VEL
LIN {X 0,Y 153.939,Z 709.673,A -85,B 0,C 180,E1 -27561.558,E2 -27561.558} C_VEL
LIN {X 0,Y 146.387,Z 721.49,A -85,B 0,C 180,E1 -27563.35,E2 -27563.35} C_VEL
LIN {X 0,Y 138.178,Z 732.445,A -85,B 0,C 180,E1 -27565.484,E2 -27565.484} C_VEL
LIN {X 0,Y 129.521,Z 742.533,A -85,B 0,C 180,E1 -27568.157,E2 -27568.157} C_VEL
LIN {X 0,Y 119.8,Z 752.398,A -85,B 0,C 180,E1 -27571.752,E2 -27571.752} C_VEL
LIN {X 0,Y 110.834,Z 760.548,A -85,B 0,C 180,E1 -27576.063,E2 -27576.063} C_VEL
LIN {X 0,Y 102.296,Z 767.312,A -85,B 0,C 180,E1 -27580.921,E2 -27580.921} C_VEL
LIN {X 0,Y 93.77,Z 773.579,A -85,B 0,C 180,E1 -27587.591,E2 -27587.591} C_VEL
LIN {X 0,Y 86.701,Z 778.42,A -85,B 0,C 180,E1 -27595.439,E2 -27595.439} C_VEL
LIN {X 0,Y 81.238,Z 781.965,A -85,B 0,C 180,E1 -27604.379,E2 -27604.379} C_VEL
LIN {X 0,Y 77.931,Z 784.305,A -85,B 0,C 180,E1 -27614.312,E2 -27614.312} C_VEL
LIN {X 0,Y 76.621,Z 785.492,A -85,B 0,C 180,E1 -27624.745,E2 -27624.745} C_VEL
LIN {X 0,Y 76.673,Z 785.649,A -85,B 0,C 180,E1 -27630.008,E2 -27630.008} C_VEL
LIN {X 0,Y 77.044,Z 785.068,A -85,B 0,C 180,E1 -27640.52,E2 -27640.52} C_VEL
LIN {X 0,Y 79.308,Z 783.344,A -85,B 0,C 180,E1 -27650.769,E2 -27650.769} C_VEL
LIN {X 0,Y 83.735,Z 780.441,A -85,B 0,C 180,E1 -27660.246,E2 -27660.246} C_VEL
LIN {X 0,Y 89.946,Z 776.292,A -85,B 0,C 180,E1 -27668.697,E2 -27668.697} C_VEL
LIN {X 0,Y 97.812,Z 770.796,A -85,B 0,C 180,E1 -27675.941,E2 -27675.941} C_VEL
LIN {X 0,Y 107.023,Z 763.801,A -85,B 0,C 180,E1 -27682.009,E2 -27682.009} C_VEL
LIN {X 0,Y 115.836,Z 756.298,A -85,B 0,C 180,E1 -27686.545,E2 -27686.545} C_VEL
LIN {X 0,Y 125.258,Z 747.255,A -85,B 0,C 180,E1 -27690.43,E2 -27690.43} C_VEL
LIN {X 0,Y 133.772,Z 738.028,A -85,B 0,C 180,E1 -27693.278,E2 -27693.278} C_VEL
LIN {X 0,Y 136.676,Z 734.56,A -85,B 0,C 180,E1 -27694.149,E2 -27694.149} C_VEL
LIN {X 0,Y 137.076,Z 733.37,A -85,B 0,C 180,E1 -27694.949,E2 -27694.949} C_VEL
LIN {X 0,Y 123.471,Z 738.979,A -85,B 0,C 180,E1 -27703.465,E2 -27703.465} C_VEL
LIN {X 0,Y 116.9,Z 742.035,A -85,B 0,C 180,E1 -27709.609,E2 -27709.609} C_VEL
LIN {X 0,Y 109.806,Z 746.524,A -85,B 0,C 180,E1 -27723.669,E2 -27723.669} C_VEL
LIN {X 0,Y 109.327,Z 748.336,A -85,B 0,C 180,E1 -27731.119,E2 -27731.119} C_VEL
LIN {X 0,Y 114.864,Z 750.915,A -85,B 0,C 180,E1 -27745.359,E2 -27745.359} C_VEL
LIN {X 0,Y 119.819,Z 751.615,A -85,B 0,C 180,E1 -27750.879,E2 -27750.879} C_VEL
LIN {X 0,Y 118.908,Z 753.15,A -85,B 0,C 180,E1 -27752.136,E2 -27752.136} C_VEL
LIN {X 0,Y 109.587,Z 761.477,A -85,B 0,C 180,E1 -27756.704,E2 -27756.704} C_VEL
LIN {X 0,Y 102.331,Z 767.179,A -85,B 0,C 180,E1 -27760.925,E2 -27760.925} C_VEL
LIN {X 0,Y 93.783,Z 773.409,A -85,B 0,C 180,E1 -27767.58,E2 -27767.58} C_VEL
LIN {X 0,Y 86.669,Z 778.22,A -85,B 0,C 180,E1 -27775.406,E2 -27775.406} C_VEL
LIN {X 0,Y 81.265,Z 781.74,A -85,B 0,C 180,E1 -27784.371,E2 -27784.371} C_VEL
LIN {X 0,Y 78.004,Z 784.049,A -85,B 0,C 180,E1 -27794.31,E2 -27794.31} C_VEL
LIN {X 0,Y 76.711,Z 785.202,A -85,B 0,C 180,E1 -27804.735,E2 -27804.735} C_VEL
LIN {X 0,Y 76.732,Z 785.35,A -85,B 0,C 180,E1 -27809.992,E2 -27809.992} C_VEL
LIN {X 0,Y 77.115,Z 784.748,A -85,B 0,C 180,E1 -27820.494,E2 -27820.494} C_VEL
LIN {X 0,Y 79.364,Z 782.997,A -85,B 0,C 180,E1 -27830.737,E2 -27830.737} C_VEL
LIN {X 0,Y 83.744,Z 780.071,A -85,B 0,C 180,E1 -27840.225,E2 -27840.225} C_VEL
LIN {X 0,Y 89.994,Z 775.898,A -85,B 0,C 180,E1 -27848.654,E2 -27848.654} C_VEL
LIN {X 0,Y 97.855,Z 770.366,A -85,B 0,C 180,E1 -27855.897,E2 -27855.897} C_VEL
LIN {X 0,Y 107.028,Z 763.325,A -85,B 0,C 180,E1 -27861.987,E2 -27861.987} C_VEL
LIN {X 0,Y 114.541,Z 756.962,A -85,B 0,C 180,E1 -27865.917,E2 -27865.917} C_VEL
LIN {X 0,Y 122.493,Z 749.434,A -85,B 0,C 180,E1 -27869.375,E2 -27869.375} C_VEL
LIN {X 0,Y 123.956,Z 747.997,A -85,B 0,C 180,E1 -27869.94,E2 -27869.94} C_VEL
LIN {X 0,Y 127.173,Z 744.359,A -85,B 0,C 180,E1 -27871.466,E2 -27871.466} C_VEL
LIN {X 0,Y 134.798,Z 733.216,A -85,B 0,C 180,E1 -27876.578,E2 -27876.578} C_VEL
LIN {X 0,Y 137.768,Z 729.081,A -85,B 0,C 180,E1 -27877.849,E2 -27877.849} C_VEL
LIN {X 0,Y 138.887,Z 727.622,A -85,B 0,C 180,E1 -27878.162,E2 -27878.162} C_VEL
LIN {X 0,Y 147.574,Z 715.529,A -85,B 0,C 180,E1 -27880.132,E2 -27880.132} C_VEL
LIN {X 0,Y 154.807,Z 703.543,A -85,B 0,C 180,E1 -27881.649,E2 -27881.649} C_VEL
LIN {X 0,Y 161.717,Z 689.837,A -85,B 0,C 180,E1 -27882.942,E2 -27882.942} C_VEL
LIN {X 0,Y 167.343,Z 676.117,A -85,B 0,C 180,E1 -27883.866,E2 -27883.866} C_VEL
LIN {X 0,Y 172.196,Z 660.788,A -85,B 0,C 180,E1 -27884.613,E2 -27884.613} C_VEL
LIN {X 0,Y 175.6,Z 645.669,A -85,B 0,C 180,E1 -27885.118,E2 -27885.118} C_VEL
LIN {X 0,Y 178.095,Z 627.458,A -85,B 0,C 180,E1 -27885.526,E2 -27885.526} C_VEL
LIN {X 0,Y 185.91,Z 556.442,A -85,B 0,C 180,E1 -27887.029,E2 -27887.029} C_VEL
LIN {X 0,Y 185.912,Z 555.616,A -85,B 0,C 180,E1 -27887.168,E2 -27887.168} C_VEL
LIN {X 0,Y 184.596,Z 552.789,A -85,B 0,C 180,E1 -27889.72,E2 -27889.72} C_VEL
LIN {X 0,Y 183.092,Z 549.437,A -85,B 0,C 180,E1 -27893.941,E2 -27893.941} C_VEL
LIN {X 0,Y 182.339,Z 548.515,A -85,B 0,C 180,E1 -27897.791,E2 -27897.791} C_VEL
LIN {X 0,Y 182.208,Z 548.773,A -85,B 0,C 180,E1 -27900.829,E2 -27900.829} C_VEL
LIN {X 0,Y 182.55,Z 551.33,A -85,B 0,C 180,E1 -27904.845,E2 -27904.845} C_VEL
LIN {X 0,Y 183.473,Z 555.221,A -85,B 0,C 180,E1 -27908.536,E2 -27908.536} C_VEL
LIN {X 0,Y 184.469,Z 559.333,A -85,B 0,C 180,E1 -27911.209,E2 -27911.209} C_VEL
LIN {X 0,Y 185.362,Z 562.864,A -85,B 0,C 180,E1 -27913.115,E2 -27913.115} C_VEL
LIN {X 0,Y 176.556,Z 640.984,A -85,B 0,C 180,E1 -27914.757,E2 -27914.757} C_VEL
LIN {X 0,Y 173.451,Z 656.703,A -85,B 0,C 180,E1 -27915.253,E2 -27915.253} C_VEL
LIN {X 0,Y 169.413,Z 670.775,A -85,B 0,C 180,E1 -27915.878,E2 -27915.878} C_VEL
LIN {X 0,Y 164.143,Z 684.731,A -85,B 0,C 180,E1 -27916.677,E2 -27916.677} C_VEL
LIN {X 0,Y 157.771,Z 698.371,A -85,B 0,C 180,E1 -27917.81,E2 -27917.81} C_VEL
LIN {X 0,Y 151.015,Z 710.392,A -85,B 0,C 180,E1 -27919.148,E2 -27919.148} C_VEL
LIN {X 0,Y 142.935,Z 722.527,A -85,B 0,C 180,E1 -27920.913,E2 -27920.913} C_VEL
LIN {X 0,Y 133.76,Z 734.19,A -85,B 0,C 180,E1 -27923.163,E2 -27923.163} C_VEL
LIN {X 0,Y 124.842,Z 744.004,A -85,B 0,C 180,E1 -27925.76,E2 -27925.76} C_VEL
LIN {X 0,Y 114.532,Z 753.841,A -85,B 0,C 180,E1 -27929.4,E2 -27929.4} C_VEL
LIN {X 0,Y 105.464,Z 761.579,A -85,B 0,C 180,E1 -27933.605,E2 -27933.605} C_VEL
LIN {X 0,Y 97.748,Z 767.298,A -85,B 0,C 180,E1 -27937.743,E2 -27937.743} C_VEL
LIN {X 0,Y 88.62,Z 773.565,A -85,B 0,C 180,E1 -27944.47,E2 -27944.47} C_VEL
LIN {X 0,Y 80.917,Z 778.406,A -85,B 0,C 180,E1 -27952.567,E2 -27952.567} C_VEL
LIN {X 0,Y 74.87,Z 781.951,A -85,B 0,C 180,E1 -27962.018,E2 -27962.018} C_VEL
LIN {X 0,Y 71.097,Z 784.291,A -85,B 0,C 180,E1 -27972.759,E2 -27972.759} C_VEL
LIN {X 0,Y 69.547,Z 785.478,A -85,B 0,C 180,E1 -27984.209,E2 -27984.209} C_VEL
LIN {X 0,Y 69.573,Z 785.635,A -85,B 0,C 180,E1 -27990.009,E2 -27990.009} C_VEL
LIN {X 0,Y 70.048,Z 785.054,A -85,B 0,C 180,E1 -28001.585,E2 -28001.585} C_VEL
LIN {X 0,Y 72.658,Z 783.33,A -85,B 0,C 180,E1 -28012.771,E2 -28012.771} C_VEL
LIN {X 0,Y 77.627,Z 780.426,A -85,B 0,C 180,E1 -28022.912,E2 -28022.912} C_VEL
LIN {X 0,Y 84.486,Z 776.276,A -85,B 0,C 180,E1 -28031.729,E2 -28031.729} C_VEL
LIN {X 0,Y 92.978,Z 770.78,A -85,B 0,C 180,E1 -28039.112,E2 -28039.112} C_VEL
LIN {X 0,Y 102.795,Z 763.783,A -85,B 0,C 180,E1 -28045.138,E2 -28045.138} C_VEL
LIN {X 0,Y 112.052,Z 756.279,A -85,B 0,C 180,E1 -28049.598,E2 -28049.598} C_VEL
LIN {X 0,Y 121.898,Z 747.235,A -85,B 0,C 180,E1 -28053.345,E2 -28053.345} C_VEL
LIN {X 0,Y 127.757,Z 741.227,A -85,B 0,C 180,E1 -28055.196,E2 -28055.196} C_VEL
LIN {X 0,Y 127.899,Z 740.28,A -85,B 0,C 180,E1 -28056.174,E2 -28056.174} C_VEL
LIN {X 0,Y 111.391,Z 746.776,A -85,B 0,C 180,E1 -28069.089,E2 -28069.089} C_VEL
LIN {X 0,Y 104.098,Z 750.982,A -85,B 0,C 180,E1 -28083.871,E2 -28083.871} C_VEL
LIN {X 0,Y 103.714,Z 752.666,A -85,B 0,C 180,E1 -28091.729,E2 -28091.729} C_VEL
LIN {X 0,Y 109.648,Z 755.063,A -85,B 0,C 180,E1 -28106.658,E2 -28106.658} C_VEL
LIN {X 0,Y 112.433,Z 755.48,A -85,B 0,C 180,E1 -28110.004,E2 -28110.004} C_VEL
LIN {X 0,Y 109.439,Z 758.252,A -85,B 0,C 180,E1 -28111.681,E2 -28111.681} C_VEL
LIN {X 0,Y 100.262,Z 765.402,A -85,B 0,C 180,E1 -28116.273,E2 -28116.273} C_VEL
LIN {X 0,Y 90.801,Z 772.013,A -85,B 0,C 180,E1 -28122.658,E2 -28122.658} C_VEL
LIN {X 0,Y 83.943,Z 776.365,A -85,B 0,C 180,E1 -28128.894,E2 -28128.894} C_VEL
LIN {X 0,Y 77.661,Z 780.151,A -85,B 0,C 180,E1 -28137.104,E2 -28137.104} C_VEL
LIN {X 0,Y 72.724,Z 783.056,A -85,B 0,C 180,E1 -28147.251,E2 -28147.251} C_VEL
LIN {X 0,Y 70.114,Z 784.781,A -85,B 0,C 180,E1 -28158.426,E2 -28158.426} C_VEL
LIN {X 0,Y 69.643,Z 785.364,A -85,B 0,C 180,E1 -28169.991,E2 -28169.991} C_VEL
LIN {X 0,Y 70.109,Z 784.762,A -85,B 0,C 180,E1 -28181.556,E2 -28181.556} C_VEL
LIN {X 0,Y 72.71,Z 783.011,A -85,B 0,C 180,E1 -28192.735,E2 -28192.735} C_VEL
LIN {X 0,Y 77.646,Z 780.085,A -85,B 0,C 180,E1 -28202.883,E2 -28202.883} C_VEL
LIN {X 0,Y 84.512,Z 775.912,A -85,B 0,C 180,E1 -28211.693,E2 -28211.693} C_VEL
LIN {X 0,Y 93.008,Z 770.38,A -85,B 0,C 180,E1 -28219.07,E2 -28219.07} C_VEL
LIN {X 0,Y 102.798,Z 763.339,A -85,B 0,C 180,E1 -28225.113,E2 -28225.113} C_VEL
LIN {X 0,Y 110.578,Z 757.051,A -85,B 0,C 180,E1 -28228.965,E2 -28228.965} C_VEL
LIN {X 0,Y 120.004,Z 748.522,A -85,B 0,C 180,E1 -28232.685,E2 -28232.685} C_VEL
LIN {X 0,Y 129.255,Z 739.049,A -85,B 0,C 180,E1 -28235.595,E2 -28235.595} C_VEL
LIN {X 0,Y 138.301,Z 728.361,A -85,B 0,C 180,E1 -28238.02,E2 -28238.02} C_VEL
LIN {X 0,Y 138.887,Z 727.622,A -85,B 0,C 180,E1 -28238.162,E2 -28238.162} C_VEL
LIN {X 0,Y 141.985,Z 723.279,A -85,B 0,C 180,E1 -28239.203,E2 -28239.203} C_VEL
LIN {X 0,Y 146.073,Z 716.101,A -85,B 0,C 180,E1 -28241.396,E2 -28241.396} C_VEL
LIN {X 0,Y 149.958,Z 708.616,A -85,B 0,C 180,E1 -28243.402,E2 -28243.402} C_VEL
LIN {X 0,Y 152.632,Z 703.718,A -85,B 0,C 180,E1 -28244.164,E2 -28244.164} C_VEL
LIN {X 0,Y 159.778,Z 689.863,A -85,B 0,C 180,E1 -28245.377,E2 -28245.377} C_VEL
LIN {X 0,Y 165.513,Z 676.149,A -85,B 0,C 180,E1 -28246.225,E2 -28246.225} C_VEL
LIN {X 0,Y 170.454,Z 660.829,A -85,B 0,C 180,E1 -28246.908,E2 -28246.908} C_VEL
LIN {X 0,Y 173.83,Z 646.167,A -85,B 0,C 180,E1 -28247.367,E2 -28247.367} C_VEL
LIN {X 0,Y 176.344,Z 628.568,A -85,B 0,C 180,E1 -28247.734,E2 -28247.734} C_VEL
LIN {X 0,Y 183.879,Z 561.636,A -85,B 0,C 180,E1 -28249.07,E2 -28249.07} C_VEL
LIN {X 0,Y 183.966,Z 560.657,A -85,B 0,C 180,E1 -28249.127,E2 -28249.127} C_VEL
LIN {X 0,Y 182.216,Z 556.606,A -85,B 0,C 180,E1 -28253.912,E2 -28253.912} C_VEL
LIN {X 0,Y 181.611,Z 555.759,A -85,B 0,C 180,E1 -28256.688,E2 -28256.688} C_VEL
LIN {X 0,Y 181.338,Z 555.736,A -85,B 0,C 180,E1 -28260.464,E2 -28260.464} C_VEL
LIN {X 0,Y 181.568,Z 558.146,A -85,B 0,C 180,E1 -28264.301,E2 -28264.301} C_VEL
LIN {X 0,Y 182.303,Z 561.735,A -85,B 0,C 180,E1 -28267.755,E2 -28267.755} C_VEL
LIN {X 0,Y 183.095,Z 565.567,A -85,B 0,C 180,E1 -28270.241,E2 -28270.241} C_VEL
LIN {X 0,Y 183.412,Z 566.94,A -85,B 0,C 180,E1 -28271.046,E2 -28271.046} C_VEL
LIN {X 0,Y 175.043,Z 639.788,A -85,B 0,C 180,E1 -28272.481,E2 -28272.481} C_VEL
LIN {X 0,Y 172.126,Z 654.892,A -85,B 0,C 180,E1 -28272.902,E2 -28272.902} C_VEL
LIN {X 0,Y 168.02,Z 669.474,A -85,B 0,C 180,E1 -28273.485,E2 -28273.485} C_VEL
LIN {X 0,Y 163.074,Z 682.759,A -85,B 0,C 180,E1 -28274.163,E2 -28274.163} C_VEL
LIN {X 0,Y 156.556,Z 696.791,A -85,B 0,C 180,E1 -28275.186,E2 -28275.186} C_VEL
LIN {X 0,Y 148.825,Z 710.37,A -85,B 0,C 180,E1 -28276.549,E2 -28276.549} C_VEL
LIN {X 0,Y 140.555,Z 722.508,A -85,B 0,C 180,E1 -28278.205,E2 -28278.205} C_VEL
LIN {X 0,Y 131.118,Z 734.172,A -85,B 0,C 180,E1 -28280.295,E2 -28280.295} C_VEL
LIN {X 0,Y 121.907,Z 743.987,A -85,B 0,C 180,E1 -28282.734,E2 -28282.734} C_VEL
LIN {X 0,Y 111.342,Z 753.702,A -85,B 0,C 180,E1 -28286.133,E2 -28286.133} C_VEL
LIN {X 0,Y 101.68,Z 761.564,A -85,B 0,C 180,E1 -28290.246,E2 -28290.246} C_VEL
LIN {X 0,Y 90.982,Z 769.004,A -85,B 0,C 180,E1 -28295.811,E2 -28295.811} C_VEL
LIN {X 0,Y 81.508,Z 774.909,A -85,B 0,C 180,E1 -28302.881,E2 -28302.881} C_VEL
LIN {X 0,Y 75.368,Z 778.393,A -85,B 0,C 180,E1 -28309.263,E2 -28309.263} C_VEL
LIN {X 0,Y 68.655,Z 781.938,A -85,B 0,C 180,E1 -28319.225,E2 -28319.225} C_VEL
LIN {X 0,Y 64.299,Z 784.278,A -85,B 0,C 180,E1 -28330.869,E2 -28330.869} C_VEL
LIN {X 0,Y 62.494,Z 785.465,A -85,B 0,C 180,E1 -28343.553,E2 -28343.553} C_VEL
LIN {X 0,Y 62.49,Z 785.621,A -85,B 0,C 180,E1 -28350.01,E2 -28350.01} C_VEL
LIN {X 0,Y 63.094,Z 785.04,A -85,B 0,C 180,E1 -28362.882,E2 -28362.882} C_VEL
LIN {X 0,Y 66.118,Z 783.315,A -85,B 0,C 180,E1 -28375.172,E2 -28375.172} C_VEL
LIN {X 0,Y 71.717,Z 780.411,A -85,B 0,C 180,E1 -28386.024,E2 -28386.024} C_VEL
LIN {X 0,Y 79.287,Z 776.26,A -85,B 0,C 180,E1 -28395.174,E2 -28395.174} C_VEL
LIN {X 0,Y 88.467,Z 770.763,A -85,B 0,C 180,E1 -28402.612,E2 -28402.612} C_VEL
LIN {X 0,Y 96.16,Z 765.67,A -85,B 0,C 180,E1 -28407.203,E2 -28407.203} C_VEL
LIN {X 0,Y 105.778,Z 758.529,A -85,B 0,C 180,E1 -28411.695,E2 -28411.695} C_VEL
LIN {X 0,Y 115.874,Z 749.937,A -85,B 0,C 180,E1 -28415.487,E2 -28415.487} C_VEL
LIN {X 0,Y 117.894,Z 748.122,A -85,B 0,C 180,E1 -28416.125,E2 -28416.125} C_VEL
LIN {X 0,Y 119.383,Z 746.337,A -85,B 0,C 180,E1 -28417.119,E2 -28417.119} C_VEL
LIN {X 0,Y 108.895,Z 750.055,A -85,B 0,C 180,E1 -28425.039,E2 -28425.039} C_VEL
LIN {X 0,Y 100.934,Z 753.339,A -85,B 0,C 180,E1 -28436.007,E2 -28436.007} C_VEL
LIN {X 0,Y 97.733,Z 756.042,A -85,B 0,C 180,E1 -28448.269,E2 -28448.269} C_VEL
LIN {X 0,Y 104.344,Z 758.974,A -85,B 0,C 180,E1 -28468.13,E2 -28468.13} C_VEL
LIN {X 0,Y 104.46,Z 759.378,A -85,B 0,C 180,E1 -28468.988,E2 -28468.988} C_VEL
LIN {X 0,Y 93.568,Z 767.213,A -85,B 0,C 180,E1 -28474.277,E2 -28474.277} C_VEL
LIN {X 0,Y 83.778,Z 773.441,A -85,B 0,C 180,E1 -28480.965,E2 -28480.965} C_VEL
LIN {X 0,Y 75.335,Z 778.251,A -85,B 0,C 180,E1 -28489.219,E2 -28489.219} C_VEL
LIN {X 0,Y 68.673,Z 781.77,A -85,B 0,C 180,E1 -28499.213,E2 -28499.213} C_VEL
LIN {X 0,Y 64.375,Z 784.077,A -85,B 0,C 180,E1 -28510.872,E2 -28510.872} C_VEL
LIN {X 0,Y 62.555,Z 785.23,A -85,B 0,C 180,E1 -28523.539,E2 -28523.539} C_VEL
LIN {X 0,Y 62.543,Z 785.378,A -85,B 0,C 180,E1 -28529.99,E2 -28529.99} C_VEL
LIN {X 0,Y 63.145,Z 784.776,A -85,B 0,C 180,E1 -28542.851,E2 -28542.851} C_VEL
LIN {X 0,Y 66.165,Z 783.025,A -85,B 0,C 180,E1 -28555.132,E2 -28555.132} C_VEL
LIN {X 0,Y 71.734,Z 780.098,A -85,B 0,C 180,E1 -28565.992,E2 -28565.992} C_VEL
LIN {X 0,Y 79.319,Z 775.926,A -85,B 0,C 180,E1 -28575.128,E2 -28575.128} C_VEL
LIN {X 0,Y 88.487,Z 770.394,A -85,B 0,C 180,E1 -28582.571,E2 -28582.571} C_VEL
LIN {X 0,Y 96.177,Z 765.279,A -85,B 0,C 180,E1 -28587.163,E2 -28587.163} C_VEL
LIN {X 0,Y 105.731,Z 758.128,A -85,B 0,C 180,E1 -28591.663,E2 -28591.663} C_VEL
LIN {X 0,Y 114.386,Z 750.806,A -85,B 0,C 180,E1 -28594.978,E2 -28594.978} C_VEL
LIN {X 0,Y 124.944,Z 740.677,A -85,B 0,C 180,E1 -28598.127,E2 -28598.127} C_VEL
LIN {X 0,Y 134.21,Z 730.308,A -85,B 0,C 180,E1 -28600.474,E2 -28600.474} C_VEL
LIN {X 0,Y 142.917,Z 719.026,A -85,B 0,C 180,E1 -28602.305,E2 -28602.305} C_VEL
LIN {X 0,Y 151.341,Z 705.965,A -85,B 0,C 180,E1 -28603.942,E2 -28603.942} C_VEL
LIN {X 0,Y 152.632,Z 703.718,A -85,B 0,C 180,E1 -28604.164,E2 -28604.164} C_VEL
LIN {X 0,Y 155.211,Z 698.776,A -85,B 0,C 180,E1 -28604.882,E2 -28604.882} C_VEL
LIN {X 0,Y 158.609,Z 690.644,A -85,B 0,C 180,E1 -28606.572,E2 -28606.572} C_VEL
LIN {X 0,Y 161.701,Z 682.276,A -85,B 0,C 180,E1 -28608.105,E2 -28608.105} C_VEL
LIN {X 0,Y 163.689,Z 676.914,A -85,B 0,C 180,E1 -28608.601,E2 -28608.601} C_VEL
LIN {X 0,Y 168.779,Z 661.611,A -85,B 0,C 180,E1 -28609.226,E2 -28609.226} C_VEL
LIN {X 0,Y 172.495,Z 645.836,A -85,B 0,C 180,E1 -28609.672,E2 -28609.672} C_VEL
LIN {X 0,Y 175.125,Z 627.367,A -85,B 0,C 180,E1 -28610.025,E2 -28610.025} C_VEL
LIN {X 0,Y 182.139,Z 566.284,A -85,B 0,C 180,E1 -28611.178,E2 -28611.178} C_VEL
LIN {X 0,Y 181.947,Z 565.493,A -85,B 0,C 180,E1 -28611.797,E2 -28611.797} C_VEL
LIN {X 0,Y 181.141,Z 563.3,A -85,B 0,C 180,E1 -28614.713,E2 -28614.713} C_VEL
LIN {X 0,Y 180.607,Z 562.628,A -85,B 0,C 180,E1 -28617.77,E2 -28617.77} C_VEL
LIN {X 0,Y 180.462,Z 562.94,A -85,B 0,C 180,E1 -28620.7,E2 -28620.7} C_VEL
LIN {X 0,Y 180.653,Z 565.344,A -85,B 0,C 180,E1 -28624.183,E2 -28624.183} C_VEL
LIN {X 0,Y 181.189,Z 568.512,A -85,B 0,C 180,E1 -28627.102,E2 -28627.102} C_VEL
LIN {X 0,Y 181.678,Z 571.238,A -85,B 0,C 180,E1 -28628.933,E2 -28628.933} C_VEL
LIN {X 0,Y 173.588,Z 640.102,A -85,B 0,C 180,E1 -28630.199,E2 -28630.199} C_VEL
LIN {X 0,Y 170.68,Z 654.841,A -85,B 0,C 180,E1 -28630.576,E2 -28630.576} C_VEL
LIN {X 0,Y 166.502,Z 669.436,A -85,B 0,C 180,E1 -28631.098,E2 -28631.098} C_VEL
LIN {X 0,Y 161.48,Z 682.729,A -85,B 0,C 180,E1 -28631.714,E2 -28631.714} C_VEL
LIN {X 0,Y 154.843,Z 696.766,A -85,B 0,C 180,E1 -28632.642,E2 -28632.642} C_VEL
LIN {X 0,Y 146.959,Z 710.348,A -85,B 0,C 180,E1 -28633.892,E2 -28633.892} C_VEL
LIN {X 0,Y 138.496,Z 722.488,A -85,B 0,C 180,E1 -28635.407,E2 -28635.407} C_VEL
LIN {X 0,Y 128.812,Z 734.155,A -85,B 0,C 180,E1 -28637.311,E2 -28637.311} C_VEL
LIN {X 0,Y 119.334,Z 743.971,A -85,B 0,C 180,E1 -28639.577,E2 -28639.577} C_VEL
LIN {X 0,Y 108.545,Z 753.564,A -85,B 0,C 180,E1 -28642.7,E2 -28642.7} C_VEL
LIN {X 0,Y 98.277,Z 761.549,A -85,B 0,C 180,E1 -28646.648,E2 -28646.648} C_VEL
LIN {X 0,Y 86.986,Z 768.99,A -85,B 0,C 180,E1 -28651.983,E2 -28651.983} C_VEL
LIN {X 0,Y 76.812,Z 774.895,A -85,B 0,C 180,E1 -28658.962,E2 -28658.962} C_VEL
LIN {X 0,Y 70.088,Z 778.379,A -85,B 0,C 180,E1 -28665.432,E2 -28665.432} C_VEL
LIN {X 0,Y 62.613,Z 781.924,A -85,B 0,C 180,E1 -28675.872,E2 -28675.872} C_VEL
LIN {X 0,Y 57.59,Z 784.264,A -85,B 0,C 180,E1 -28688.537,E2 -28688.537} C_VEL
LIN {X 0,Y 55.438,Z 785.451,A -85,B 0,C 180,E1 -28702.728,E2 -28702.728} C_VEL
LIN {X 0,Y 55.39,Z 785.608,A -85,B 0,C 180,E1 -28710.011,E2 -28710.011} C_VEL
LIN {X 0,Y 56.156,Z 785.026,A -85,B 0,C 180,E1 -28724.507,E2 -28724.507} C_VEL
LIN {X 0,Y 59.722,Z 783.3,A -85,B 0,C 180,E1 -28738.092,E2 -28738.092} C_VEL
LIN {X 0,Y 66.056,Z 780.396,A -85,B 0,C 180,E1 -28749.682,E2 -28749.682} C_VEL
LIN {X 0,Y 74.409,Z 776.244,A -85,B 0,C 180,E1 -28759.09,E2 -28759.09} C_VEL
LIN {X 0,Y 84.302,Z 770.747,A -85,B 0,C 180,E1 -28766.49,E2 -28766.49} C_VEL
LIN {X 0,Y 95.344,Z 763.748,A -85,B 0,C 180,E1 -28772.208,E2 -28772.208} C_VEL
LIN {X 0,Y 105.231,Z 756.49,A -85,B 0,C 180,E1 -28776.207,E2 -28776.207} C_VEL
LIN {X 0,Y 108.705,Z 753.662,A -85,B 0,C 180,E1 -28777.402,E2 -28777.402} C_VEL
LIN {X 0,Y 110.024,Z 752.208,A -85,B 0,C 180,E1 -28778.574,E2 -28778.574} C_VEL
LIN {X 0,Y 99.854,Z 755.52,A -85,B 0,C 180,E1 -28787.81,E2 -28787.81} C_VEL
LIN {X 0,Y 91.911,Z 759.481,A -85,B 0,C 180,E1 -28806.2,E2 -28806.2} C_VEL
LIN {X 0,Y 94.428,Z 761.674,A -85,B 0,C 180,E1 -28821.847,E2 -28821.847} C_VEL
LIN {X 0,Y 96.84,Z 762.258,A -85,B 0,C 180,E1 -28826.608,E2 -28826.608} C_VEL
LIN {X 0,Y 95.402,Z 763.529,A -85,B 0,C 180,E1 -28827.858,E2 -28827.858} C_VEL
LIN {X 0,Y 87.022,Z 768.932,A -85,B 0,C 180,E1 -28831.994,E2 -28831.994} C_VEL
LIN {X 0,Y 76.823,Z 774.798,A -85,B 0,C 180,E1 -28838.947,E2 -28838.947} C_VEL
LIN {X 0,Y 70.059,Z 778.267,A -85,B 0,C 180,E1 -28845.384,E2 -28845.384} C_VEL
LIN {X 0,Y 62.652,Z 781.784,A -85,B 0,C 180,E1 -28855.872,E2 -28855.872} C_VEL
LIN {X 0,Y 57.66,Z 784.092,A -85,B 0,C 180,E1 -28868.541,E2 -28868.541} C_VEL
LIN {X 0,Y 55.489,Z 785.244,A -85,B 0,C 180,E1 -28882.712,E2 -28882.712} C_VEL
LIN {X 0,Y 55.461,Z 785.391,A -85,B 0,C 180,E1 -28889.989,E2 -28889.989} C_VEL
LIN {X 0,Y 56.232,Z 784.789,A -85,B 0,C 180,E1 -28904.464,E2 -28904.464} C_VEL
LIN {X 0,Y 59.763,Z 783.038,A -85,B 0,C 180,E1 -28918.047,E2 -28918.047} C_VEL
LIN {X 0,Y 66.072,Z 780.112,A -85,B 0,C 180,E1 -28929.646,E2 -28929.646} C_VEL
LIN {X 0,Y 74.436,Z 775.94,A -85,B 0,C 180,E1 -28939.04,E2 -28939.04} C_VEL
LIN {X 0,Y 84.334,Z 770.408,A -85,B 0,C 180,E1 -28946.43,E2 -28946.43} C_VEL
LIN {X 0,Y 92.497,Z 765.293,A -85,B 0,C 180,E1 -28950.886,E2 -28950.886} C_VEL
LIN {X 0,Y 101.113,Z 759.219,A -85,B 0,C 180,E1 -28954.617,E2 -28954.617} C_VEL
LIN {X 0,Y 110.018,Z 752.156,A -85,B 0,C 180,E1 -28957.844,E2 -28957.844} C_VEL
LIN {X 0,Y 120.904,Z 742.303,A -85,B 0,C 180,E1 -28960.82,E2 -28960.82} C_VEL
LIN {X 0,Y 130.402,Z 732.206,A -85,B 0,C 180,E1 -28963.045,E2 -28963.045} C_VEL
LIN {X 0,Y 140.107,Z 720.179,A -85,B 0,C 180,E1 -28964.911,E2 -28964.911} C_VEL
LIN {X 0,Y 148.647,Z 707.477,A -85,B 0,C 180,E1 -28966.42,E2 -28966.42} C_VEL
LIN {X 0,Y 156.481,Z 693.361,A -85,B 0,C 180,E1 -28967.627,E2 -28967.627} C_VEL
LIN {X 0,Y 162.719,Z 679.492,A -85,B 0,C 180,E1 -28968.469,E2 -28968.469} C_VEL
LIN {X 0,Y 163.689,Z 676.914,A -85,B 0,C 180,E1 -28968.601,E2 -28968.601} C_VEL
LIN {X 0,Y 165.591,Z 671.465,A -85,B 0,C 180,E1 -28969.041,E2 -28969.041} C_VEL
LIN {X 0,Y 167.94,Z 662.602,A -85,B 0,C 180,E1 -28970.34,E2 -28970.34} C_VEL
LIN {X 0,Y 169.872,Z 653.584,A -85,B 0,C 180,E1 -28971.576,E2 -28971.576} C_VEL
LIN {X 0,Y 170.981,Z 647.892,A -85,B 0,C 180,E1 -28971.956,E2 -28971.956} C_VEL
LIN {X 0,Y 173.332,Z 633.473,A -85,B 0,C 180,E1 -28972.213,E2 -28972.213} C_VEL
LIN {X 0,Y 180.593,Z 571.485,A -85,B 0,C 180,E1 -28973.296,E2 -28973.296} C_VEL
LIN {X 0,Y 180.093,Z 570.071,A -85,B 0,C 180,E1 -28975.524,E2 -28975.524} C_VEL
LIN {X 0,Y 179.743,Z 569.667,A -85,B 0,C 180,E1 -28977.759,E2 -28977.759} C_VEL
LIN {X 0,Y 179.591,Z 569.957,A -85,B 0,C 180,E1 -28980.469,E2 -28980.469} C_VEL
LIN {X 0,Y 179.697,Z 572.263,A -85,B 0,C 180,E1 -28983.714,E2 -28983.714} C_VEL
LIN {X 0,Y 180.078,Z 575.063,A -85,B 0,C 180,E1 -28986.302,E2 -28986.302} C_VEL
LIN {X 0,Y 180.172,Z 575.727,A -85,B 0,C 180,E1 -28986.784,E2 -28986.784} C_VEL
LIN {X 0,Y 172.514,Z 639.763,A -85,B 0,C 180,E1 -28987.878,E2 -28987.878} C_VEL
LIN {X 0,Y 169.522,Z 654.792,A -85,B 0,C 180,E1 -28988.22,E2 -28988.22} C_VEL
LIN {X 0,Y 165.283,Z 669.4,A -85,B 0,C 180,E1 -28988.686,E2 -28988.686} C_VEL
LIN {X 0,Y 160.192,Z 682.699,A -85,B 0,C 180,E1 -28989.233,E2 -28989.233} C_VEL
LIN {X 0,Y 153.444,Z 696.741,A -85,B 0,C 180,E1 -28990.052,E2 -28990.052} C_VEL
LIN {X 0,Y 145.535,Z 710.133,A -85,B 0,C 180,E1 -28991.138,E2 -28991.138} C_VEL
LIN {X 0,Y 136.779,Z 722.469,A -85,B 0,C 180,E1 -28992.534,E2 -28992.534} C_VEL
LIN {X 0,Y 126.872,Z 734.137,A -85,B 0,C 180,E1 -28994.233,E2 -28994.233} C_VEL
LIN {X 0,Y 117.141,Z 743.955,A -85,B 0,C 180,E1 -28996.294,E2 -28996.294} C_VEL
LIN {X 0,Y 105.992,Z 753.548,A -85,B 0,C 180,E1 -28999.133,E2 -28999.133} C_VEL
LIN {X 0,Y 95.289,Z 761.535,A -85,B 0,C 180,E1 -29002.809,E2 -29002.809} C_VEL
LIN {X 0,Y 83.421,Z 768.976,A -85,B 0,C 180,E1 -29007.815,E2 -29007.815} C_VEL
LIN {X 0,Y 72.518,Z 774.881,A -85,B 0,C 180,E1 -29014.552,E2 -29014.552} C_VEL
LIN {X 0,Y 65.175,Z 778.365,A -85,B 0,C 180,E1 -29021.005,E2 -29021.005} C_VEL
LIN {X 0,Y 56.835,Z 781.91,A -85,B 0,C 180,E1 -29031.824,E2 -29031.824} C_VEL
LIN {X 0,Y 51.011,Z 784.25,A -85,B 0,C 180,E1 -29045.6,E2 -29045.6} C_VEL
LIN {X 0,Y 48.388,Z 785.437,A -85,B 0,C 180,E1 -29061.662,E2 -29061.662} C_VEL
LIN {X 0,Y 48.304,Z 785.594,A -85,B 0,C 180,E1 -29070.013,E2 -29070.013} C_VEL
LIN {X 0,Y 49.286,Z 785.011,A -85,B 0,C 180,E1 -29086.583,E2 -29086.583} C_VEL
LIN {X 0,Y 53.516,Z 783.286,A -85,B 0,C 180,E1 -29101.701,E2 -29101.701} C_VEL
LIN {X 0,Y 60.715,Z 780.381,A -85,B 0,C 180,E1 -29114.003,E2 -29114.003} C_VEL
LIN {X 0,Y 69.936,Z 776.229,A -85,B 0,C 180,E1 -29123.521,E2 -29123.521} C_VEL
LIN {X 0,Y 80.567,Z 770.73,A -85,B 0,C 180,E1 -29130.743,E2 -29130.743} C_VEL
LIN {X 0,Y 92.227,Z 763.73,A -85,B 0,C 180,E1 -29136.141,E2 -29136.141} C_VEL
LIN {X 0,Y 100.09,Z 758.272,A -85,B 0,C 180,E1 -29139.062,E2 -29139.062} C_VEL
LIN {X 0,Y 101.208,Z 757.369,A -85,B 0,C 180,E1 -29139.683,E2 -29139.683} C_VEL
LIN {X 0,Y 91.028,Z 760.448,A -85,B 0,C 180,E1 -29151.117,E2 -29151.117} C_VEL
LIN {X 0,Y 85.611,Z 763.602,A -85,B 0,C 180,E1 -29169.864,E2 -29169.864} C_VEL
LIN {X 0,Y 88.657,Z 765.172,A -85,B 0,C 180,E1 -29183.35,E2 -29183.35} C_VEL
LIN {X 0,Y 88.789,Z 765.745,A -85,B 0,C 180,E1 -29185.318,E2 -29185.318} C_VEL
LIN {X 0,Y 77.871,Z 772.061,A -85,B 0,C 180,E1 -29190.96,E2 -29190.96} C_VEL
LIN {X 0,Y 67.36,Z 777.282,A -85,B 0,C 180,E1 -29198.756,E2 -29198.756} C_VEL
LIN {X 0,Y 60.743,Z 780.196,A -85,B 0,C 180,E1 -29206.022,E2 -29206.022} C_VEL
LIN {X 0,Y 53.573,Z 783.1,A -85,B 0,C 180,E1 -29218.336,E2 -29218.336} C_VEL
LIN {X 0,Y 49.358,Z 784.824,A -85,B 0,C 180,E1 -29233.441,E2 -29233.441} C_VEL
LIN {X 0,Y 48.36,Z 785.405,A -85,B 0,C 180,E1 -29249.987,E2 -29249.987} C_VEL
LIN {X 0,Y 49.35,Z 784.803,A -85,B 0,C 180,E1 -29266.535,E2 -29266.535} C_VEL
LIN {X 0,Y 53.556,Z 783.052,A -85,B 0,C 180,E1 -29281.648,E2 -29281.648} C_VEL
LIN {X 0,Y 60.728,Z 780.126,A -85,B 0,C 180,E1 -29293.962,E2 -29293.962} C_VEL
LIN {X 0,Y 69.948,Z 775.953,A -85,B 0,C 180,E1 -29303.479,E2 -29303.479} C_VEL
LIN {X 0,Y 80.587,Z 770.422,A -85,B 0,C 180,E1 -29310.687,E2 -29310.687} C_VEL
LIN {X 0,Y 89.241,Z 765.307,A -85,B 0,C 180,E1 -29314.894,E2 -29314.894} C_VEL
LIN {X 0,Y 98.241,Z 759.234,A -85,B 0,C 180,E1 -29318.415,E2 -29318.415} C_VEL
LIN {X 0,Y 107.527,Z 752.172,A -85,B 0,C 180,E1 -29321.372,E2 -29321.372} C_VEL
LIN {X 0,Y 118.748,Z 742.319,A -85,B 0,C 180,E1 -29324.078,E2 -29324.078} C_VEL
LIN {X 0,Y 128.503,Z 732.224,A -85,B 0,C 180,E1 -29326.09,E2 -29326.09} C_VEL
LIN {X 0,Y 138.423,Z 720.198,A -85,B 0,C 180,E1 -29327.76,E2 -29327.76} C_VEL
LIN {X 0,Y 146.879,Z 707.901,A -85,B 0,C 180,E1 -29329.077,E2 -29329.077} C_VEL
LIN {X 0,Y 154.273,Z 695.001,A -85,B 0,C 180,E1 -29330.082,E2 -29330.082} C_VEL
LIN {X 0,Y 161.029,Z 680.542,A -85,B 0,C 180,E1 -29330.886,E2 -29330.886} C_VEL
LIN {X 0,Y 166.535,Z 665.329,A -85,B 0,C 180,E1 -29331.499,E2 -29331.499} C_VEL
LIN {X 0,Y 170.655,Z 649.548,A -85,B 0,C 180,E1 -29331.934,E2 -29331.934} C_VEL
LIN {X 0,Y 170.981,Z 647.892,A -85,B 0,C 180,E1 -29331.956,E2 -29331.956} C_VEL
LIN {X 0,Y 171.984,Z 642.15,A -85,B 0,C 180,E1 -29332.306,E2 -29332.306} C_VEL
LIN {X 0,Y 173.79,Z 623.534,A -85,B 0,C 180,E1 -29334.497,E2 -29334.497} C_VEL
LIN {X 0,Y 174.402,Z 617.732,A -85,B 0,C 180,E1 -29334.811,E2 -29334.811} C_VEL
LIN {X 0,Y 179.235,Z 577.182,A -85,B 0,C 180,E1 -29335.452,E2 -29335.452} C_VEL
LIN {X 0,Y 178.879,Z 576.712,A -85,B 0,C 180,E1 -29337.749,E2 -29337.749} C_VEL
LIN {X 0,Y 178.715,Z 577.093,A -85,B 0,C 180,E1 -29340.471,E2 -29340.471} C_VEL
LIN {X 0,Y 178.794,Z 579.634,A -85,B 0,C 180,E1 -29343.733,E2 -29343.733} C_VEL
LIN {X 0,Y 178.891,Z 580.437,A -85,B 0,C 180,E1 -29344.579,E2 -29344.579} C_VEL
LIN {X 0,Y 171.876,Z 638.43,A -85,B 0,C 180,E1 -29345.513,E2 -29345.513} C_VEL
LIN {X 0,Y 168.867,Z 653.861,A -85,B 0,C 180,E1 -29345.807,E2 -29345.807} C_VEL
LIN {X 0,Y 164.363,Z 669.364,A -85,B 0,C 180,E1 -29346.243,E2 -29346.243} C_VEL
LIN {X 0,Y 159.209,Z 682.67,A -85,B 0,C 180,E1 -29346.715,E2 -29346.715} C_VEL
LIN {X 0,Y 153.221,Z 695.162,A -85,B 0,C 180,E1 -29347.335,E2 -29347.335} C_VEL
LIN {X 0,Y 145.589,Z 708.222,A -85,B 0,C 180,E1 -29348.207,E2 -29348.207} C_VEL
LIN {X 0,Y 137.105,Z 720.338,A -85,B 0,C 180,E1 -29349.367,E2 -29349.367} C_VEL
LIN {X 0,Y 126.988,Z 732.358,A -85,B 0,C 180,E1 -29350.809,E2 -29350.809} C_VEL
LIN {X 0,Y 116.991,Z 742.451,A -85,B 0,C 180,E1 -29352.557,E2 -29352.557} C_VEL
LIN {X 0,Y 105.491,Z 752.304,A -85,B 0,C 180,E1 -29355.006,E2 -29355.006} C_VEL
LIN {X 0,Y 94.318,Z 760.475,A -85,B 0,C 180,E1 -29358.209,E2 -29358.209} C_VEL
LIN {X 0,Y 83.361,Z 767.241,A -85,B 0,C 180,E1 -29361.991,E2 -29361.991} C_VEL
LIN {X 0,Y 71.531,Z 773.51,A -85,B 0,C 180,E1 -29367.86,E2 -29367.86} C_VEL
LIN {X 0,Y 60.716,Z 778.351,A -85,B 0,C 180,E1 -29375.897,E2 -29375.897} C_VEL
LIN {X 0,Y 51.407,Z 781.896,A -85,B 0,C 180,E1 -29386.894,E2 -29386.894} C_VEL
LIN {X 0,Y 44.612,Z 784.236,A -85,B 0,C 180,E1 -29401.813,E2 -29401.813} C_VEL
LIN {X 0,Y 41.373,Z 785.423,A -85,B 0,C 180,E1 -29420.235,E2 -29420.235} C_VEL
LIN {X 0,Y 41.19,Z 785.58,A -85,B 0,C 180,E1 -29430.015,E2 -29430.015} C_VEL
LIN {X 0,Y 42.511,Z 784.997,A -85,B 0,C 180,E1 -29449.323,E2 -29449.323} C_VEL
LIN {X 0,Y 47.578,Z 783.271,A -85,B 0,C 180,E1 -29466.233,E2 -29466.233} C_VEL
LIN {X 0,Y 55.786,Z 780.366,A -85,B 0,C 180,E1 -29479.119,E2 -29479.119} C_VEL
LIN {X 0,Y 65.927,Z 776.213,A -85,B 0,C 180,E1 -29488.537,E2 -29488.537} C_VEL
LIN {X 0,Y 77.322,Z 770.714,A -85,B 0,C 180,E1 -29495.375,E2 -29495.375} C_VEL
LIN {X 0,Y 89.577,Z 763.713,A -85,B 0,C 180,E1 -29500.322,E2 -29500.322} C_VEL
LIN {X 0,Y 91.253,Z 762.304,A -85,B 0,C 180,E1 -29502.057,E2 -29502.057} C_VEL
LIN {X 0,Y 80.691,Z 765.617,A -85,B 0,C 180,E1 -29519.999,E2 -29519.999} C_VEL
LIN {X 0,Y 79.813,Z 767.462,A -85,B 0,C 180,E1 -29535.317,E2 -29535.317} C_VEL
LIN {X 0,Y 81.453,Z 768.08,A -85,B 0,C 180,E1 -29541.619,E2 -29541.619} C_VEL
LIN {X 0,Y 79.793,Z 769.27,A -85,B 0,C 180,E1 -29543.571,E2 -29543.571} C_VEL
LIN {X 0,Y 68.737,Z 774.829,A -85,B 0,C 180,E1 -29549.631,E2 -29549.631} C_VEL
LIN {X 0,Y 60.686,Z 778.298,A -85,B 0,C 180,E1 -29555.823,E2 -29555.823} C_VEL
LIN {X 0,Y 51.432,Z 781.814,A -85,B 0,C 180,E1 -29566.887,E2 -29566.887} C_VEL
LIN {X 0,Y 44.668,Z 784.12,A -85,B 0,C 180,E1 -29581.819,E2 -29581.819} C_VEL
LIN {X 0,Y 41.415,Z 785.271,A -85,B 0,C 180,E1 -29600.215,E2 -29600.215} C_VEL
LIN {X 0,Y 41.274,Z 785.419,A -85,B 0,C 180,E1 -29609.985,E2 -29609.985} C_VEL
LIN {X 0,Y 42.565,Z 784.817,A -85,B 0,C 180,E1 -29629.267,E2 -29629.267} C_VEL
LIN {X 0,Y 47.614,Z 783.066,A -85,B 0,C 180,E1 -29646.17,E2 -29646.17} C_VEL
LIN {X 0,Y 55.797,Z 780.139,A -85,B 0,C 180,E1 -29659.072,E2 -29659.072} C_VEL
LIN {X 0,Y 65.943,Z 775.967,A -85,B 0,C 180,E1 -29668.478,E2 -29668.478} C_VEL
LIN {X 0,Y 77.332,Z 770.436,A -85,B 0,C 180,E1 -29675.32,E2 -29675.32} C_VEL
LIN {X 0,Y 89.577,Z 763.397,A -85,B 0,C 180,E1 -29680.281,E2 -29680.281} C_VEL
LIN {X 0,Y 100.01,Z 756.303,A -85,B 0,C 180,E1 -29683.675,E2 -29683.675} C_VEL
LIN {X 0,Y 110.38,Z 748.171,A -85,B 0,C 180,E1 -29686.136,E2 -29686.136} C_VEL
LIN {X 0,Y 121.975,Z 737.504,A -85,B 0,C 180,E1 -29688.353,E2 -29688.353} C_VEL
LIN {X 0,Y 132.029,Z 726.504,A -85,B 0,C 180,E1 -29689.954,E2 -29689.954} C_VEL
LIN {X 0,Y 141.32,Z 714.451,A -85,B 0,C 180,E1 -29691.232,E2 -29691.232} C_VEL
LIN {X 0,Y 149.794,Z 701.204,A -85,B 0,C 180,E1 -29692.328,E2 -29692.328} C_VEL
LIN {X 0,Y 156.629,Z 688.21,A -85,B 0,C 180,E1 -29693.061,E2 -29693.061} C_VEL
LIN {X 0,Y 162.629,Z 674.043,A -85,B 0,C 180,E1 -29693.648,E2 -29693.648} C_VEL
LIN {X 0,Y 167.358,Z 659.482,A -85,B 0,C 180,E1 -29694.069,E2 -29694.069} C_VEL
LIN {X 0,Y 170.807,Z 644.522,A -85,B 0,C 180,E1 -29694.399,E2 -29694.399} C_VEL
LIN {X 0,Y 173.613,Z 624.399,A -85,B 0,C 180,E1 -29694.691,E2 -29694.691} C_VEL
LIN {X 0,Y 174.402,Z 617.732,A -85,B 0,C 180,E1 -29694.811,E2 -29694.811} C_VEL
LIN {X 0,Y 175.033,Z 611.939,A -85,B 0,C 180,E1 -29695.127,E2 -29695.127} C_VEL
LIN {X 0,Y 176.9,Z 593.325,A -85,B 0,C 180,E1 -29697.259,E2 -29697.259} C_VEL
LIN {X 0,Y 177.572,Z 587.532,A -85,B 0,C 180,E1 -29697.558,E2 -29697.558} C_VEL
LIN {X 0,Y 178.022,Z 583.778,A -85,B 0,C 180,E1 -29697.651,E2 -29697.651} C_VEL
LIN {X 0,Y 177.845,Z 584.129,A -85,B 0,C 180,E1 -29700.237,E2 -29700.237} C_VEL
LIN {X 0,Y 177.817,Z 585.731,A -85,B 0,C 180,E1 -29702.421,E2 -29702.421} C_VEL
LIN {X 0,Y 170.95,Z 640.889,A -85,B 0,C 180,E1 -29703.182,E2 -29703.182} C_VEL
LIN {X 0,Y 167.648,Z 656.458,A -85,B 0,C 180,E1 -29703.468,E2 -29703.468} C_VEL
LIN {X 0,Y 162.875,Z 671.859,A -85,B 0,C 180,E1 -29703.84,E2 -29703.84} C_VEL
LIN {X 0,Y 156.8,Z 686.532,A -85,B 0,C 180,E1 -29704.294,E2 -29704.294} C_VEL
LIN {X 0,Y 149.884,Z 699.807,A -85,B 0,C 180,E1 -29704.919,E2 -29704.919} C_VEL
LIN {X 0,Y 142.387,Z 711.69,A -85,B 0,C 180,E1 -29705.666,E2 -29705.666} C_VEL
LIN {X 0,Y 133.552,Z 723.488,A -85,B 0,C 180,E1 -29706.696,E2 -29706.696} C_VEL
LIN {X 0,Y 124.138,Z 734.102,A -85,B 0,C 180,E1 -29707.841,E2 -29707.841} C_VEL
LIN {X 0,Y 113.962,Z 743.923,A -85,B 0,C 180,E1 -29709.389,E2 -29709.389} C_VEL
LIN {X 0,Y 102.206,Z 753.518,A -85,B 0,C 180,E1 -29711.548,E2 -29711.548} C_VEL
LIN {X 0,Y 92.325,Z 760.461,A -85,B 0,C 180,E1 -29713.968,E2 -29713.968} C_VEL
LIN {X 0,Y 80.957,Z 767.226,A -85,B 0,C 180,E1 -29717.297,E2 -29717.297} C_VEL
LIN {X 0,Y 68.481,Z 773.496,A -85,B 0,C 180,E1 -29722.56,E2 -29722.56} C_VEL
LIN {X 0,Y 56.806,Z 778.338,A -85,B 0,C 180,E1 -29730.021,E2 -29730.021} C_VEL
LIN {X 0,Y 46.449,Z 781.883,A -85,B 0,C 180,E1 -29740.863,E2 -29740.863} C_VEL
LIN {X 0,Y 38.461,Z 784.223,A -85,B 0,C 180,E1 -29756.777,E2 -29756.777} C_VEL
LIN {X 0,Y 34.378,Z 785.409,A -85,B 0,C 180,E1 -29778.222,E2 -29778.222} C_VEL
LIN {X 0,Y 34.083,Z 785.566,A -85,B 0,C 180,E1 -29790.018,E2 -29790.018} C_VEL
LIN {X 0,Y 35.85,Z 784.983,A -85,B 0,C 180,E1 -29813.103,E2 -29813.103} C_VEL
LIN {X 0,Y 42.024,Z 783.257,A -85,B 0,C 180,E1 -29832.006,E2 -29832.006} C_VEL
LIN {X 0,Y 51.387,Z 780.351,A -85,B 0,C 180,E1 -29845.165,E2 -29845.165} C_VEL
LIN {X 0,Y 62.485,Z 776.197,A -85,B 0,C 180,E1 -29854.153,E2 -29854.153} C_VEL
LIN {X 0,Y 74.627,Z 770.697,A -85,B 0,C 180,E1 -29860.37,E2 -29860.37} C_VEL
LIN {X 0,Y 80.951,Z 767.396,A -85,B 0,C 180,E1 -29862.769,E2 -29862.769} C_VEL
LIN {X 0,Y 82.168,Z 766.525,A -85,B 0,C 180,E1 -29864.084,E2 -29864.084} C_VEL
LIN {X 0,Y 73.155,Z 769.473,A -85,B 0,C 180,E1 -29885.512,E2 -29885.512} C_VEL
LIN {X 0,Y 73.786,Z 770.587,A -85,B 0,C 180,E1 -29897.707,E2 -29897.707} C_VEL
LIN {X 0,Y 73.113,Z 771.376,A -85,B 0,C 180,E1 -29900.388,E2 -29900.388} C_VEL
LIN {X 0,Y 62.529,Z 776.077,A -85,B 0,C 180,E1 -29905.929,E2 -29905.929} C_VEL
LIN {X 0,Y 51.408,Z 780.227,A -85,B 0,C 180,E1 -29914.868,E2 -29914.868} C_VEL
LIN {X 0,Y 42.07,Z 783.129,A -85,B 0,C 180,E1 -29928.051,E2 -29928.051} C_VEL
LIN {X 0,Y 35.931,Z 784.852,A -85,B 0,C 180,E1 -29946.953,E2 -29946.953} C_VEL
LIN {X 0,Y 34.16,Z 785.433,A -85,B 0,C 180,E1 -29969.982,E2 -29969.982} C_VEL
LIN {X 0,Y 35.921,Z 784.831,A -85,B 0,C 180,E1 -29993.016,E2 -29993.016} C_VEL
LIN {X 0,Y 42.051,Z 783.079,A -85,B 0,C 180,E1 -30011.932,E2 -30011.932} C_VEL
LIN {X 0,Y 51.394,Z 780.153,A -85,B 0,C 180,E1 -30025.11,E2 -30025.11} C_VEL
LIN {X 0,Y 62.504,Z 775.981,A -85,B 0,C 180,E1 -30034.072,E2 -30034.072} C_VEL
LIN {X 0,Y 74.629,Z 770.45,A -85,B 0,C 180,E1 -30040.317,E2 -30040.317} C_VEL
LIN {X 0,Y 87.424,Z 763.411,A -85,B 0,C 180,E1 -30044.696,E2 -30044.696} C_VEL
LIN {X 0,Y 98.305,Z 756.271,A -85,B 0,C 180,E1 -30047.688,E2 -30047.688} C_VEL
LIN {X 0,Y 110.583,Z 746.781,A -85,B 0,C 180,E1 -30050.057,E2 -30050.057} C_VEL
LIN {X 0,Y 120.737,Z 737.521,A -85,B 0,C 180,E1 -30051.672,E2 -30051.672} C_VEL
LIN {X 0,Y 131.833,Z 725.518,A -85,B 0,C 180,E1 -30053.12,E2 -30053.12} C_VEL
LIN {X 0,Y 141.267,Z 713.267,A -85,B 0,C 180,E1 -30054.215,E2 -30054.215} C_VEL
LIN {X 0,Y 149.876,Z 699.72,A -85,B 0,C 180,E1 -30055.117,E2 -30055.117} C_VEL
LIN {X 0,Y 156.796,Z 686.438,A -85,B 0,C 180,E1 -30055.725,E2 -30055.725} C_VEL
LIN {X 0,Y 162.866,Z 671.749,A -85,B 0,C 180,E1 -30056.209,E2 -30056.209} C_VEL
LIN {X 0,Y 167.426,Z 657.2,A -85,B 0,C 180,E1 -30056.546,E2 -30056.546} C_VEL
LIN {X 0,Y 170.701,Z 642.278,A -85,B 0,C 180,E1 -30056.822,E2 -30056.822} C_VEL
LIN {X 0,Y 173.952,Z 617.437,A -85,B 0,C 180,E1 -30057.146,E2 -30057.146} C_VEL
LIN {X 0,Y 177.572,Z 587.532,A -85,B 0,C 180,E1 -30057.558,E2 -30057.558} C_VEL
LIN {X 0,Y 177.407,Z 588.533,A -85,B 0,C 180,E1 -30057.92,E2 -30057.92} C_VEL
LIN {X 0,Y 176.73,Z 593.607,A -85,B 0,C 180,E1 -30058.509,E2 -30058.509} C_VEL
LIN {X 0,Y 175.086,Z 606.652,A -85,B 0,C 180,E1 -30059.262,E2 -30059.262} C_VEL
LIN {X 0,Y 174.366,Z 612.47,A -85,B 0,C 180,E1 -30059.449,E2 -30059.449} C_VEL
LIN {X 0,Y 173.648,Z 618.311,A -85,B 0,C 180,E1 -30059.47,E2 -30059.47} C_VEL
LIN {X 0,Y 170.425,Z 642.53,A -85,B 0,C 180,E1 -30059.199,E2 -30059.199} C_VEL
LIN {X 0,Y 166.929,Z 658.083,A -85,B 0,C 180,E1 -30058.961,E2 -30058.961} C_VEL
LIN {X 0,Y 162.113,Z 673.005,A -85,B 0,C 180,E1 -30058.678,E2 -30058.678} C_VEL
LIN {X 0,Y 156.428,Z 686.467,A -85,B 0,C 180,E1 -30058.315,E2 -30058.315} C_VEL
LIN {X 0,Y 149.439,Z 699.744,A -85,B 0,C 180,E1 -30057.829,E2 -30057.829} C_VEL
LIN {X 0,Y 140.726,Z 713.287,A -85,B 0,C 180,E1 -30057.11,E2 -30057.11} C_VEL
LIN {X 0,Y 131.171,Z 725.536,A -85,B 0,C 180,E1 -30056.208,E2 -30056.208} C_VEL
LIN {X 0,Y 119.912,Z 737.537,A -85,B 0,C 180,E1 -30055.041,E2 -30055.041} C_VEL
LIN {X 0,Y 107.857,Z 748.203,A -85,B 0,C 180,E1 -30053.503,E2 -30053.503} C_VEL
LIN {X 0,Y 95.428,Z 757.368,A -85,B 0,C 180,E1 -30051.53,E2 -30051.53} C_VEL
LIN {X 0,Y 82.468,Z 765.35,A -85,B 0,C 180,E1 -30048.492,E2 -30048.492} C_VEL
LIN {X 0,Y 69.276,Z 771.995,A -85,B 0,C 180,E1 -30044.494,E2 -30044.494} C_VEL
LIN {X 0,Y 59.722,Z 775.995,A -85,B 0,C 180,E1 -30040.259,E2 -30040.259} C_VEL
LIN {X 0,Y 47.666,Z 780.167,A -85,B 0,C 180,E1 -30032.18,E2 -30032.18} C_VEL
LIN {X 0,Y 37.043,Z 783.093,A -85,B 0,C 180,E1 -30019.341,E2 -30019.341} C_VEL
LIN {X 0,Y 29.481,Z 784.844,A -85,B 0,C 180,E1 -29998.451,E2 -29998.451} C_VEL
LIN {X 0,Y 27.052,Z 785.447,A -85,B 0,C 180,E1 -29969.977,E2 -29969.977} C_VEL
LIN {X 0,Y 29.493,Z 784.866,A -85,B 0,C 180,E1 -29941.513,E2 -29941.513} C_VEL
LIN {X 0,Y 37.063,Z 783.144,A -85,B 0,C 180,E1 -29920.643,E2 -29920.643} C_VEL
LIN {X 0,Y 47.681,Z 780.242,A -85,B 0,C 180,E1 -29907.798,E2 -29907.798} C_VEL
LIN {X 0,Y 59.748,Z 776.093,A -85,B 0,C 180,E1 -29899.748,E2 -29899.748} C_VEL
LIN {X 0,Y 66.086,Z 773.522,A -85,B 0,C 180,E1 -29896.809,E2 -29896.809} C_VEL
LIN {X 0,Y 66.476,Z 772.845,A -85,B 0,C 180,E1 -29892.206,E2 -29892.206} C_VEL
LIN {X 0,Y 69.408,Z 771.219,A -85,B 0,C 180,E1 -29874.188,E2 -29874.188} C_VEL
LIN {X 0,Y 71.931,Z 770.556,A -85,B 0,C 180,E1 -29868.731,E2 -29868.731} C_VEL
LIN {X 0,Y 72.536,Z 770.681,A -85,B 0,C 180,E1 -29865.703,E2 -29865.703} C_VEL
LIN {X 0,Y 59.708,Z 776.182,A -85,B 0,C 180,E1 -29860.36,E2 -29860.36} C_VEL
LIN {X 0,Y 47.662,Z 780.336,A -85,B 0,C 180,E1 -29852.246,E2 -29852.246} C_VEL
LIN {X 0,Y 37.026,Z 783.242,A -85,B 0,C 180,E1 -29839.423,E2 -29839.423} C_VEL
LIN {X 0,Y 29.424,Z 784.969,A -85,B 0,C 180,E1 -29818.56,E2 -29818.56} C_VEL
LIN {X 0,Y 26.99,Z 785.552,A -85,B 0,C 180,E1 -29790.023,E2 -29790.023} C_VEL
LIN {X 0,Y 29.418,Z 784.944,A -85,B 0,C 180,E1 -29761.482,E2 -29761.482} C_VEL
LIN {X 0,Y 37.026,Z 783.185,A -85,B 0,C 180,E1 -29740.629,E2 -29740.629} C_VEL
LIN {X 0,Y 47.681,Z 780.252,A -85,B 0,C 180,E1 -29727.854,E2 -29727.854} C_VEL
LIN {X 0,Y 59.733,Z 776.072,A -85,B 0,C 180,E1 -29719.769,E2 -29719.769} C_VEL
LIN {X 0,Y 72.54,Z 770.535,A -85,B 0,C 180,E1 -29714.378,E2 -29714.378} C_VEL
LIN {X 0,Y 82.478,Z 765.416,A -85,B 0,C 180,E1 -29711.543,E2 -29711.543} C_VEL
LIN {X 0,Y 92.534,Z 759.339,A -85,B 0,C 180,E1 -29709.167,E2 -29709.167} C_VEL
LIN {X 0,Y 104.433,Z 750.938,A -85,B 0,C 180,E1 -29707.015,E2 -29707.015} C_VEL
LIN {X 0,Y 116.461,Z 740.81,A -85,B 0,C 180,E1 -29705.372,E2 -29705.372} C_VEL
LIN {X 0,Y 126.836,Z 730.443,A -85,B 0,C 180,E1 -29704.222,E2 -29704.222} C_VEL
LIN {X 0,Y 137.034,Z 718.305,A -85,B 0,C 180,E1 -29703.287,E2 -29703.287} C_VEL
LIN {X 0,Y 144.82,Z 707.325,A -85,B 0,C 180,E1 -29702.556,E2 -29702.556} C_VEL
LIN {X 0,Y 152.934,Z 693.502,A -85,B 0,C 180,E1 -29701.946,E2 -29701.946} C_VEL
LIN {X 0,Y 159.49,Z 679.655,A -85,B 0,C 180,E1 -29701.515,E2 -29701.515} C_VEL
LIN {X 0,Y 164.742,Z 665.485,A -85,B 0,C 180,E1 -29701.21,E2 -29701.21} C_VEL
LIN {X 0,Y 169.005,Z 649.696,A -85,B 0,C 180,E1 -29700.94,E2 -29700.94} C_VEL
LIN {X 0,Y 171.642,Z 634.663,A -85,B 0,C 180,E1 -29700.763,E2 -29700.763} C_VEL
LIN {X 0,Y 176.961,Z 591.317,A -85,B 0,C 180,E1 -29700.202,E2 -29700.202} C_VEL
LIN {X 0,Y 176.987,Z 591.091,A -85,B 0,C 180,E1 -29699.858,E2 -29699.858} C_VEL
LIN {X 0,Y 173.648,Z 618.311,A -85,B 0,C 180,E1 -29699.47,E2 -29699.47} C_VEL
LIN {X 0,Y 173.633,Z 618.568,A -85,B 0,C 180,E1 -29699.468,E2 -29699.468} C_VEL
LIN {X 0,Y 173.633,Z 725.625,A -85,B 0,C 180,E1 -29699.468,E2 -29699.468} C_VEL
LIN {X 0,Y 145.792,Z 725.625,A -85,B 0,C 180,E1 -29699.626,E2 -29699.626} C_VEL
LIN {X 0,Y 143.793,Z 723.625,A -85,B 0,C 180,E1 -29699.64,E2 -29699.64} C_VEL
LIN {X 0,Y 143.793,Z 714.852,A -85,B 0,C 180,E1 -29699.64,E2 -29699.64} C_VEL
LIN {X 0,Y 140.32,Z 713.634,A -85,B 0,C 180,E1 -29700,E2 -29700} C_VEL
LIN {X 0,Y 131.771,Z 724.507,A -85,B 0,C 180,E1 -29700.641,E2 -29700.641} C_VEL
LIN {X 0,Y 121.257,Z 735.832,A -85,B 0,C 180,E1 -29701.397,E2 -29701.397} C_VEL
LIN {X 0,Y 110.774,Z 745.362,A -85,B 0,C 180,E1 -29702.377,E2 -29702.377} C_VEL
LIN {X 0,Y 98.59,Z 754.708,A -85,B 0,C 180,E1 -29703.744,E2 -29703.744} C_VEL
LIN {X 0,Y 88.225,Z 761.476,A -85,B 0,C 180,E1 -29705.371,E2 -29705.371} C_VEL
LIN {X 0,Y 77.916,Z 767.198,A -85,B 0,C 180,E1 -29707.231,E2 -29707.231} C_VEL
LIN {X 0,Y 64.357,Z 773.468,A -85,B 0,C 180,E1 -29710.69,E2 -29710.69} C_VEL
LIN {X 0,Y 51.165,Z 778.31,A -85,B 0,C 180,E1 -29715.993,E2 -29715.993} C_VEL
LIN {X 0,Y 38.641,Z 781.855,A -85,B 0,C 180,E1 -29724.62,E2 -29724.62} C_VEL
LIN {X 0,Y 27.633,Z 784.195,A -85,B 0,C 180,E1 -29740.307,E2 -29740.307} C_VEL
LIN {X 0,Y 20.633,Z 785.382,A -85,B 0,C 180,E1 -29770.118,E2 -29770.118} C_VEL
LIN {X 0,Y 19.884,Z 785.538,A -85,B 0,C 180,E1 -29790.031,E2 -29790.031} C_VEL
LIN {X 0,Y 23.415,Z 784.955,A -85,B 0,C 180,E1 -29826.924,E2 -29826.924} C_VEL
LIN {X 0,Y 32.835,Z 783.228,A -85,B 0,C 180,E1 -29848.925,E2 -29848.925} C_VEL
LIN {X 0,Y 44.78,Z 780.32,A -85,B 0,C 180,E1 -29860.372,E2 -29860.372} C_VEL
LIN {X 0,Y 57.697,Z 776.166,A -85,B 0,C 180,E1 -29867.068,E2 -29867.068} C_VEL
LIN {X 0,Y 64.357,Z 773.591,A -85,B 0,C 180,E1 -29869.418,E2 -29869.418} C_VEL
LIN {X 0,Y 59.792,Z 775.257,A -85,B 0,C 180,E1 -29891.109,E2 -29891.109} C_VEL
LIN {X 0,Y 57.721,Z 776.109,A -85,B 0,C 180,E1 -29893.035,E2 -29893.035} C_VEL
LIN {X 0,Y 44.796,Z 780.257,A -85,B 0,C 180,E1 -29899.683,E2 -29899.683} C_VEL
LIN {X 0,Y 32.861,Z 783.158,A -85,B 0,C 180,E1 -29911.152,E2 -29911.152} C_VEL
LIN {X 0,Y 23.473,Z 784.88,A -85,B 0,C 180,E1 -29933.182,E2 -29933.182} C_VEL
LIN {X 0,Y 19.959,Z 785.461,A -85,B 0,C 180,E1 -29969.969,E2 -29969.969} C_VEL
LIN {X 0,Y 23.459,Z 784.858,A -85,B 0,C 180,E1 -30006.778,E2 -30006.778} C_VEL
LIN {X 0,Y 32.841,Z 783.107,A -85,B 0,C 180,E1 -30028.834,E2 -30028.834} C_VEL
LIN {X 0,Y 44.778,Z 780.18,A -85,B 0,C 180,E1 -30040.297,E2 -30040.297} C_VEL
LIN {X 0,Y 57.696,Z 776.008,A -85,B 0,C 180,E1 -30046.978,E2 -30046.978} C_VEL
LIN {X 0,Y 71.099,Z 770.478,A -85,B 0,C 180,E1 -30051.232,E2 -30051.232} C_VEL
LIN {X 0,Y 84.778,Z 763.44,A -85,B 0,C 180,E1 -30054.07,E2 -30054.07} C_VEL
LIN {X 0,Y 97.033,Z 755.77,A -85,B 0,C 180,E1 -30056.116,E2 -30056.116} C_VEL
LIN {X 0,Y 109.029,Z 746.812,A -85,B 0,C 180,E1 -30057.454,E2 -30057.454} C_VEL
LIN {X 0,Y 119.507,Z 737.554,A -85,B 0,C 180,E1 -30058.457,E2 -30058.457} C_VEL
LIN {X 0,Y 130.893,Z 725.555,A -85,B 0,C 180,E1 -30059.327,E2 -30059.327} C_VEL
LIN {X 0,Y 140.32,Z 713.634,A -85,B 0,C 180,E1 -30060,E2 -30060} C_VEL
LIN {X 0,Y 143.846,Z 714.842,A -85,B 0,C 180,E1 -30060.28,E2 -30060.28} C_VEL
LIN {X 0,Y 143.846,Z 768.409,A -85,B 0,C 180,E1 -30060.28,E2 -30060.28} C_VEL
LIN {X 0,Y 97.666,Z 768.409,A -85,B 0,C 180,E1 -30059.534,E2 -30059.534} C_VEL
LIN {X 0,Y 95.668,Z 766.409,A -85,B 0,C 180,E1 -30059.485,E2 -30059.485} C_VEL
LIN {X 0,Y 95.668,Z 760.138,A -85,B 0,C 180,E1 -30059.485,E2 -30059.485} C_VEL
LIN {X 0,Y 92.754,Z 758.426,A -85,B 0,C 180,E1 -30060,E2 -30060} C_VEL
LIN {X 0,Y 84.342,Z 763.462,A -85,B 0,C 180,E1 -30061.182,E2 -30061.182} C_VEL
LIN {X 0,Y 70.364,Z 770.507,A -85,B 0,C 180,E1 -30062.994,E2 -30062.994} C_VEL
LIN {X 0,Y 56.518,Z 776.045,A -85,B 0,C 180,E1 -30065.964,E2 -30065.964} C_VEL
LIN {X 0,Y 42.906,Z 780.225,A -85,B 0,C 180,E1 -30070.722,E2 -30070.722} C_VEL
LIN {X 0,Y 29.775,Z 783.158,A -85,B 0,C 180,E1 -30079.304,E2 -30079.304} C_VEL
LIN {X 0,Y 18.2,Z 784.917,A -85,B 0,C 180,E1 -30099.494,E2 -30099.494} C_VEL
LIN {X 0,Y 12.772,Z 785.524,A -85,B 0,C 180,E1 -30150.049,E2 -30150.049} C_VEL
LIN {X 0,Y 18.211,Z 784.941,A -85,B 0,C 180,E1 -30200.574,E2 -30200.574} C_VEL
LIN {X 0,Y 29.786,Z 783.213,A -85,B 0,C 180,E1 -30220.76,E2 -30220.76} C_VEL
LIN {X 0,Y 42.911,Z 780.305,A -85,B 0,C 180,E1 -30229.398,E2 -30229.398} C_VEL
LIN {X 0,Y 52.352,Z 777.558,A -85,B 0,C 180,E1 -30232.99,E2 -30232.99} C_VEL
LIN {X 0,Y 55.229,Z 776.577,A -85,B 0,C 180,E1 -30234.909,E2 -30234.909} C_VEL
LIN {X 0,Y 53.454,Z 777.12,A -85,B 0,C 180,E1 -30243.688,E2 -30243.688} C_VEL
LIN {X 0,Y 51.697,Z 777.737,A -85,B 0,C 180,E1 -30247.331,E2 -30247.331} C_VEL
LIN {X 0,Y 36.27,Z 781.873,A -85,B 0,C 180,E1 -30254.27,E2 -30254.27} C_VEL
LIN {X 0,Y 23.685,Z 784.178,A -85,B 0,C 180,E1 -30267.048,E2 -30267.048} C_VEL
LIN {X 0,Y 14.207,Z 785.327,A -85,B 0,C 180,E1 -30300.3,E2 -30300.3} C_VEL
LIN {X 0,Y 12.853,Z 785.475,A -85,B 0,C 180,E1 -30329.951,E2 -30329.951} C_VEL
LIN {X 0,Y 18.257,Z 784.872,A -85,B 0,C 180,E1 -30380.289,E2 -30380.289} C_VEL
LIN {X 0,Y 29.781,Z 783.12,A -85,B 0,C 180,E1 -30400.662,E2 -30400.662} C_VEL
LIN {X 0,Y 42.901,Z 780.194,A -85,B 0,C 180,E1 -30409.312,E2 -30409.312} C_VEL
LIN {X 0,Y 56.516,Z 776.022,A -85,B 0,C 180,E1 -30414.056,E2 -30414.056} C_VEL
LIN {X 0,Y 70.364,Z 770.493,A -85,B 0,C 180,E1 -30417.014,E2 -30417.014} C_VEL
LIN {X 0,Y 84.339,Z 763.455,A -85,B 0,C 180,E1 -30418.917,E2 -30418.917} C_VEL
LIN {X 0,Y 92.754,Z 758.426,A -85,B 0,C 180,E1 -30420,E2 -30420} C_VEL
LIN {X 0,Y 95.758,Z 760.127,A -85,B 0,C 180,E1 -30420.33,E2 -30420.33} C_VEL
LIN {X 0,Y 95.758,Z 788.411,A -85,B 0,C 180,E1 -30420.33,E2 -30420.33} C_VEL
LIN {X 0,Y 52.228,Z 788.411,A -85,B 0,C 180,E1 -30419.647,E2 -30419.647} C_VEL
LIN {X 0,Y 50.229,Z 786.411,A -85,B 0,C 180,E1 -30419.587,E2 -30419.587} C_VEL
LIN {X 0,Y 50.229,Z 780.65,A -85,B 0,C 180,E1 -30419.587,E2 -30419.587} C_VEL
LIN {X 0,Y 47.743,Z 778.717,A -85,B 0,C 180,E1 -30420.001,E2 -30420.001} C_VEL
LIN {X 0,Y 35.173,Z 781.828,A -85,B 0,C 180,E1 -30422.89,E2 -30422.89} C_VEL
LIN {X 0,Y 21.372,Z 784.168,A -85,B 0,C 180,E1 -30429.605,E2 -30429.605} C_VEL
LIN {X 0,Y 8.71,Z 785.354,A -85,B 0,C 180,E1 -30456.331,E2 -30456.331} C_VEL
LIN {X 0,Y 5.673,Z 785.511,A -85,B 0,C 180,E1 -30510.11,E2 -30510.11} C_VEL
LIN {X 0,Y 14.743,Z 784.926,A -85,B 0,C 180,E1 -30582.579,E2 -30582.579} C_VEL
LIN {X 0,Y 28.25,Z 783.198,A -85,B 0,C 180,E1 -30594.548,E2 -30594.548} C_VEL
LIN {X 0,Y 42.185,Z 780.29,A -85,B 0,C 180,E1 -30599.01,E2 -30599.01} C_VEL
LIN {X 0,Y 47.018,Z 779.033,A -85,B 0,C 180,E1 -30599.999,E2 -30599.999} C_VEL
LIN {X 0,Y 35.195,Z 781.888,A -85,B 0,C 180,E1 -30602.889,E2 -30602.889} C_VEL
LIN {X 0,Y 21.402,Z 784.192,A -85,B 0,C 180,E1 -30609.722,E2 -30609.722} C_VEL
LIN {X 0,Y 8.773,Z 785.341,A -85,B 0,C 180,E1 -30636.649,E2 -30636.649} C_VEL
LIN {X 0,Y 5.741,Z 785.488,A -85,B 0,C 180,E1 -30689.891,E2 -30689.891} C_VEL
LIN {X 0,Y 14.751,Z 784.886,A -85,B 0,C 180,E1 -30762.202,E2 -30762.202} C_VEL
LIN {X 0,Y 28.233,Z 783.134,A -85,B 0,C 180,E1 -30774.452,E2 -30774.452} C_VEL
LIN {X 0,Y 42.164,Z 780.208,A -85,B 0,C 180,E1 -30778.92,E2 -30778.92} C_VEL
LIN {X 0,Y 47.743,Z 778.717,A -85,B 0,C 180,E1 -30780.001,E2 -30780.001} C_VEL
LIN {X 0,Y 47.743,Z 778.717,A -85,B 0,C 180,E1 -30780.001,E2 -30780.001}

QRS_NEXT_CUT()

QRS_NEXT()
QRS_HOME()

END
